(* Logix 5000 project; controller Close_Palletizing 1769-L33ERM rev 33.13; software revision 33.00 *)

TASK MainTask (continuous, watchdog 500 ms) : MainProgram

MODULES
   Local : 1769-L33ERM (Compact 0, rev 33.13)
      BrazingOvenEthernetCard : 1756-ENBT (Ethernet 192.168.1.100, rev 5.1, Output RPI 10 ms)
         BrazingOvenPLC : vendor 1 type 14 code 92 (ICP 0, rev 23.12, $5738e604$ RPI 20 ms, $87ed6ff7$ RPI 20 ms)
      Fanuc_5 : ETHERNET-MODULE (Ethernet 192.168.1.5, rev 1.1, Output RPI 10 ms)
           Fanuc_5:O.Data[3].1   // *Hold
           Fanuc_5:O.Data[0]   // Part Width to give to Fanuc
           Fanuc_5:O.Data[2]   // Part Length to give to Fanuc
           Fanuc_5:O.Data[3].0   // *IMSTP
           Fanuc_5:O.Data[1]   // Part ID to give to Fanuc
           Fanuc_5:O.Data[3].2   // *SFSPD
           Fanuc_5:O.Data[3].3   // Cycle stop
           Fanuc_5:O.Data[3].4   // Fault reset
           Fanuc_5:O.Data[3].5   // Start
           Fanuc_5:O.Data[3].6   // Home
           Fanuc_5:O.Data[3].7   // Enable
           Fanuc_5:O.Data[3].8   // PNS strobe
           Fanuc_5:O.Data[3].9   // Prod start
           Fanuc_5:I.Data[2].0   // Cmd enabled
           Fanuc_5:I.Data[2].1   // System ready
           Fanuc_5:I.Data[2].2   // Prg running
           Fanuc_5:I.Data[2].3   // Prg paused
           Fanuc_5:I.Data[2].4   // Motion held
           Fanuc_5:I.Data[2].5   // Fault
           Fanuc_5:I.Data[2].6   // At perch
           Fanuc_5:I.Data[2].7   // TP enabled
           Fanuc_5:I.Data[2].8   // Batt alarm
           Fanuc_5:I.Data[2].9   // Busy
           Fanuc_5:I.Data[2].10   // ACK1/SNO1
           Fanuc_5:I.Data[2].11   // ACK2/SNO2
           Fanuc_5:I.Data[2].12   // ACK3/SNO3
           Fanuc_5:I.Data[2].13   // ACK4/SNO4
           Fanuc_5:I.Data[2].14   // ACK5/SNO5
           Fanuc_5:I.Data[2].15   // ACK6/SNO6
           Fanuc_5:I.Data[3].2   // SNACK
           Fanuc_5:I.Data[3].0   // ACK7/SNO7
           Fanuc_5:I.Data[3].1   // ACK8/SNO8
           Fanuc_5:I.Data[3].3   // Reserved
      YRC1000_Rbt_Ctlr : ETHERNET-MODULE (Ethernet 192.168.1.41, rev 1.1, Output RPI 10 ms)
      IFM_Module_Fence : vendor 322 type 12 code 1120 (Ethernet 192.168.1.43, rev 1.5, StandardDataDriven RPI 10 ms)
           IFM_Module_Fence:I1.Data[0].0   // Port 1 Pin 4
           IFM_Module_Fence:I1.Data[0].1   // Port 2 Pin 4
           IFM_Module_Fence:I1.Data[0].10   // Port 3 Pin 2
           IFM_Module_Fence:I1.Data[0].11   // Port 4 Pin 2
           IFM_Module_Fence:I1.Data[0].12   // Reserved
           IFM_Module_Fence:I1.Data[0].13   // Reserved
           IFM_Module_Fence:I1.Data[0].14   // Reserved
           IFM_Module_Fence:I1.Data[0].15   // Reserved
           IFM_Module_Fence:I1.Data[0].2   // Port 3 Pin 4
           IFM_Module_Fence:I1.Data[0].3   // Port 4 Pin 4
           IFM_Module_Fence:I1.Data[0].4   // Reserved
           IFM_Module_Fence:I1.Data[0].5   // Reserved
           IFM_Module_Fence:I1.Data[0].6   // Reserved
           IFM_Module_Fence:I1.Data[0].7   // Reserved
           IFM_Module_Fence:I1.Data[0].8   // Port 1 Pin 2
           IFM_Module_Fence:I1.Data[0].9   // Port 2 Pin 2
           IFM_Module_Fence:I1.Data[100]   // Port 3 Input Process Data
           IFM_Module_Fence:I1.Data[101]   // Port 3 Input Process Data
           IFM_Module_Fence:I1.Data[102]   // Port 3 Input Process Data
           IFM_Module_Fence:I1.Data[103]   // Port 3 Input Process Data
           IFM_Module_Fence:I1.Data[104]   // Port 3 Input Process Data
           IFM_Module_Fence:I1.Data[105]   // Port 3 Input Process Data
           IFM_Module_Fence:I1.Data[106]   // Port 3 Input Process Data
           IFM_Module_Fence:I1.Data[107]   // Port 4 Input Process Data
           IFM_Module_Fence:I1.Data[108]   // Port 4 Input Process Data
           IFM_Module_Fence:I1.Data[109]   // Port 4 Input Process Data
           IFM_Module_Fence:I1.Data[10]   // Command Response Or Diagnostic Data 7
           IFM_Module_Fence:I1.Data[110]   // Port 4 Input Process Data
           IFM_Module_Fence:I1.Data[111]   // Port 4 Input Process Data
           IFM_Module_Fence:I1.Data[112]   // Port 4 Input Process Data
           IFM_Module_Fence:I1.Data[113]   // Port 4 Input Process Data
           IFM_Module_Fence:I1.Data[114]   // Port 4 Input Process Data
           IFM_Module_Fence:I1.Data[115]   // Port 4 Input Process Data
           IFM_Module_Fence:I1.Data[116]   // Port 4 Input Process Data
           IFM_Module_Fence:I1.Data[117]   // Port 4 Input Process Data
           IFM_Module_Fence:I1.Data[118]   // Port 4 Input Process Data
           IFM_Module_Fence:I1.Data[119]   // Port 4 Input Process Data
           IFM_Module_Fence:I1.Data[11]   // Command Response Or Diagnostic Data 9
           IFM_Module_Fence:I1.Data[120]   // Port 4 Input Process Data
           IFM_Module_Fence:I1.Data[121]   // Port 4 Input Process Data
           IFM_Module_Fence:I1.Data[122]   // Port 4 Input Process Data
           IFM_Module_Fence:I1.Data[12]   // Command Response Or Diagnostic Data 11
           IFM_Module_Fence:I1.Data[13]   // Command Response Or Diagnostic Data 13
           IFM_Module_Fence:I1.Data[14]   // Command Response Or Diagnostic Data 15
           IFM_Module_Fence:I1.Data[15]   // Command Response Or Diagnostic Data 17
           IFM_Module_Fence:I1.Data[16]   // Command Response Or Diagnostic Data 19
           IFM_Module_Fence:I1.Data[17]   // Command Response Or Diagnostic Data 21
           IFM_Module_Fence:I1.Data[18]   // Command Response Or Diagnostic Data 23
           IFM_Module_Fence:I1.Data[19]   // Command Response Or Diagnostic Data 25
           IFM_Module_Fence:I1.Data[1]   // AL1x2x Digital Input Short/Overload Status
           IFM_Module_Fence:I1.Data[1].0   // Port 1 Short/Overload
           IFM_Module_Fence:I1.Data[1].1   // Port 2 Short/Overload
           IFM_Module_Fence:I1.Data[1].10   // Reserved
           IFM_Module_Fence:I1.Data[1].11   // Reserved
           IFM_Module_Fence:I1.Data[1].12   // Reserved
           IFM_Module_Fence:I1.Data[1].13   // Reserved
           IFM_Module_Fence:I1.Data[1].14   // Reserved
           IFM_Module_Fence:I1.Data[1].15   // Reserved
           IFM_Module_Fence:I1.Data[1].2   // Port 3 Short/Overload
           IFM_Module_Fence:I1.Data[1].3   // Port 4 Short/Overload
           IFM_Module_Fence:I1.Data[1].4   // Reserved
           IFM_Module_Fence:I1.Data[1].5   // Reserved
           IFM_Module_Fence:I1.Data[1].6   // Reserved
           IFM_Module_Fence:I1.Data[1].7   // Reserved
           IFM_Module_Fence:I1.Data[1].8   // Reserved
           IFM_Module_Fence:I1.Data[1].9   // Reserved
           IFM_Module_Fence:I1.Data[20]   // Command Response Or Diagnostic Data 27
           IFM_Module_Fence:I1.Data[21]   // Command Response Or Diagnostic Data 29
           IFM_Module_Fence:I1.Data[22]   // Command Response Or Diagnostic Data 31
           IFM_Module_Fence:I1.Data[23].0   // Port 1 IO-Link Mode
           IFM_Module_Fence:I1.Data[23].1   // Port 1 NO IO-Link Device Connected
           IFM_Module_Fence:I1.Data[23].10   // Reserved
           IFM_Module_Fence:I1.Data[23].11   // Reserved
           IFM_Module_Fence:I1.Data[23].12   // Reserved
           IFM_Module_Fence:I1.Data[23].13   // Reserved
           IFM_Module_Fence:I1.Data[23].14   // Reserved
           IFM_Module_Fence:I1.Data[23].15   // Reserved
           IFM_Module_Fence:I1.Data[23].2   // Port 1 IO-Link Data Invalid
           IFM_Module_Fence:I1.Data[23].3   // Port 1 Incorrect Vendor or Device ID
           IFM_Module_Fence:I1.Data[23].5   // Reserved
           IFM_Module_Fence:I1.Data[23].6   // Reserved
           IFM_Module_Fence:I1.Data[23].7   // Reserved
           IFM_Module_Fence:I1.Data[23].8   // Reserved
           IFM_Module_Fence:I1.Data[23].9   // Reserved
           IFM_Module_Fence:I1.Data[24]   // Port 1 Vendor ID
           IFM_Module_Fence:I1.Data[25]   // Port 1 Device ID (Low Word)
           IFM_Module_Fence:I1.Data[26]   // Port 1 Device ID (High Word)
           IFM_Module_Fence:I1.Data[0]   // AL1x2x Digital Input Status
           IFM_Module_Fence:I1.Data[27]   // Port 1 IO-Link Event Data
           IFM_Module_Fence:I1.Data[27].0   // Port 1 Event Instance
           IFM_Module_Fence:I1.Data[27].1   // Port 1 Event Instance
           IFM_Module_Fence:I1.Data[27].10   // Port 1 Event Code 1
           IFM_Module_Fence:I1.Data[27].11   // Port 1 Event Code 1
           IFM_Module_Fence:I1.Data[27].12   // Port 1 Event Code 1
           IFM_Module_Fence:I1.Data[27].13   // Port 1 Event Code 1
           IFM_Module_Fence:I1.Data[27].14   // Port 1 Event Code 1
           IFM_Module_Fence:I1.Data[27].15   // Port 1 Event Code 1
           IFM_Module_Fence:I1.Data[27].3   // Port 1 Event Source
           IFM_Module_Fence:I1.Data[27].8   // Port 1 Event Code 1
           IFM_Module_Fence:I1.Data[27].9   // Port 1 Event Code 1
           IFM_Module_Fence:I1.Data[28].0   // Port 1 Event Code 2
           IFM_Module_Fence:I1.Data[28].1   // Port 1 Event Code 2
           IFM_Module_Fence:I1.Data[28].10   // Port 1 Event Instance
           IFM_Module_Fence:I1.Data[27].2   // Port 1 Event Instance
           IFM_Module_Fence:I1.Data[28].12   // Port 1 Event Type
           IFM_Module_Fence:I1.Data[28].13   // Port 1 Event Type
           IFM_Module_Fence:I1.Data[28].14   // Port 1 Event Mode
           IFM_Module_Fence:I1.Data[28].15   // Port 1 Event Mode
           IFM_Module_Fence:I1.Data[28].2   // Port 1 Event Code 2
           IFM_Module_Fence:I1.Data[28].3   // Port 1 Event Code 2
           IFM_Module_Fence:I1.Data[28].4   // Port 1 Event Code 2
           IFM_Module_Fence:I1.Data[28].5   // Port 1 Event Code 2
           IFM_Module_Fence:I1.Data[28].6   // Port 1 Event Code 2
           IFM_Module_Fence:I1.Data[28].7   // Port 1 Event Code 2
           IFM_Module_Fence:I1.Data[28].11   // Port 1 Event Source
           IFM_Module_Fence:I1.Data[28].8   // Port 1 Event Instance
           IFM_Module_Fence:I1.Data[28].9   // Port 1 Event Instance
           IFM_Module_Fence:I1.Data[29].0   // Port 1 Event Code 1
           IFM_Module_Fence:I1.Data[29].1   // Port 1 Event Code 1
           IFM_Module_Fence:I1.Data[29]   // Port 1 IO-Link Event Data
           IFM_Module_Fence:I1.Data[29].10   // Port 1 Event Code 2
           IFM_Module_Fence:I1.Data[29].11   // Port 1 Event Code 2
           IFM_Module_Fence:I1.Data[29].12   // Port 1 Event Code 2
           IFM_Module_Fence:I1.Data[29].13   // Port 1 Event Code 2
           IFM_Module_Fence:I1.Data[29].14   // Port 1 Event Code 2
           IFM_Module_Fence:I1.Data[29].2   // Port 1 Event Code 1
           IFM_Module_Fence:I1.Data[29].3   // Port 1 Event Code 1
           IFM_Module_Fence:I1.Data[29].4   // Port 1 Event Code 1
           IFM_Module_Fence:I1.Data[29].5   // Port 1 Event Code 1
           IFM_Module_Fence:I1.Data[29].6   // Port 1 Event Code 1
           IFM_Module_Fence:I1.Data[29].7   // Port 1 Event Code 1
           IFM_Module_Fence:I1.Data[29].8   // Port 1 Event Code 2
           IFM_Module_Fence:I1.Data[29].9   // Port 1 Event Code 2
           IFM_Module_Fence:I1.Data[2]   // Port Number
           IFM_Module_Fence:I1.Data[29].15   // Port 1 Event Code 2
           IFM_Module_Fence:I1.Data[30]   // Port 1 IO-Link Event Data
           IFM_Module_Fence:I1.Data[30].0   // Port 1 Event Instance
           IFM_Module_Fence:I1.Data[30].1   // Port 1 Event Instance
           IFM_Module_Fence:I1.Data[30].10   // Port 1 Event Code 1
           IFM_Module_Fence:I1.Data[30].11   // Port 1 Event Code 1
           IFM_Module_Fence:I1.Data[30].12   // Port 1 Event Code 1
           IFM_Module_Fence:I1.Data[30].13   // Port 1 Event Code 1
           IFM_Module_Fence:I1.Data[30].14   // Port 1 Event Code 1
           IFM_Module_Fence:I1.Data[30].15   // Port 1 Event Code 1
           IFM_Module_Fence:I1.Data[30].3   // Port 1 Event Source
           IFM_Module_Fence:I1.Data[23]   // Port 1 IO Link Status
           IFM_Module_Fence:I1.Data[27].4   // Port 1 Event Type
           IFM_Module_Fence:I1.Data[27].5   // Port 1 Event Type
           IFM_Module_Fence:I1.Data[27].6   // Port 1 Event Mode
           IFM_Module_Fence:I1.Data[30].8   // Port 1 Event Code 1
           IFM_Module_Fence:I1.Data[30].9   // Port 1 Event Code 1
           IFM_Module_Fence:I1.Data[30].2   // Port 1 Event Instance
           IFM_Module_Fence:I1.Data[31].0   // Port 1 Event Code 2
           IFM_Module_Fence:I1.Data[31].1   // Port 1 Event Code 2
           IFM_Module_Fence:I1.Data[31].10   // Reserved
           IFM_Module_Fence:I1.Data[31].11   // Reserved
           IFM_Module_Fence:I1.Data[31].12   // Reserved
           IFM_Module_Fence:I1.Data[31].13   // Reserved
           IFM_Module_Fence:I1.Data[31].14   // Reserved
           IFM_Module_Fence:I1.Data[31].15   // Reserved
           IFM_Module_Fence:I1.Data[31].2   // Port 1 Event Code 2
           IFM_Module_Fence:I1.Data[31].3   // Port 1 Event Code 2
           IFM_Module_Fence:I1.Data[31].4   // Port 1 Event Code 2
           IFM_Module_Fence:I1.Data[31].5   // Port 1 Event Code 2
           IFM_Module_Fence:I1.Data[31].6   // Port 1 Event Code 2
           IFM_Module_Fence:I1.Data[31].7   // Port 1 Event Code 2
           IFM_Module_Fence:I1.Data[31].8   // Reserved
           IFM_Module_Fence:I1.Data[31].9   // Reserved
           IFM_Module_Fence:I1.Data[27].7   // Port 1 Event Mode
           IFM_Module_Fence:I1.Data[32].0   // Port 2 IO-Link Mode
           IFM_Module_Fence:I1.Data[32].1   // Port 2 NO IO-Link Device Connected
           IFM_Module_Fence:I1.Data[32].10   // Reserved
           IFM_Module_Fence:I1.Data[32].11   // Reserved
           IFM_Module_Fence:I1.Data[32].12   // Reserved
           IFM_Module_Fence:I1.Data[32].13   // Reserved
           IFM_Module_Fence:I1.Data[32].14   // Reserved
           IFM_Module_Fence:I1.Data[32].15   // Reserved
           IFM_Module_Fence:I1.Data[32].2   // Port 2 IO-Link Data Invalid
           IFM_Module_Fence:I1.Data[32].3   // Port 2 Incorrect Vendor or Device ID
           IFM_Module_Fence:I1.Data[23].4   // Port 1 IO-Link Data String Error
           IFM_Module_Fence:I1.Data[32].5   // Reserved
           IFM_Module_Fence:I1.Data[32].6   // Reserved
           IFM_Module_Fence:I1.Data[32].7   // Reserved
           IFM_Module_Fence:I1.Data[32].8   // Reserved
           IFM_Module_Fence:I1.Data[32].9   // Reserved
           IFM_Module_Fence:I1.Data[33]   // Port 2 Vendor ID
           IFM_Module_Fence:I1.Data[34]   // Port 2 Device ID (Low Word)
           IFM_Module_Fence:I1.Data[35]   // Port 2 Device ID (High Word)
           IFM_Module_Fence:I1.Data[31]   // Port 1 IO-Link Event Data
           IFM_Module_Fence:I1.Data[36]   // Port 2 IO-Link Event Data
           IFM_Module_Fence:I1.Data[36].0   // Port 2 Event Instance
           IFM_Module_Fence:I1.Data[36].1   // Port 2 Event Instance
           IFM_Module_Fence:I1.Data[36].10   // Port 2 Event Code 1
           IFM_Module_Fence:I1.Data[36].11   // Port 2 Event Code 1
           IFM_Module_Fence:I1.Data[36].12   // Port 2 Event Code 1
           IFM_Module_Fence:I1.Data[36].13   // Port 2 Event Code 1
           IFM_Module_Fence:I1.Data[36].14   // Port 2 Event Code 1
           IFM_Module_Fence:I1.Data[36].15   // Port 2 Event Code 1
           IFM_Module_Fence:I1.Data[36].3   // Port 2 Event Source
           IFM_Module_Fence:I1.Data[30].4   // Port 1 Event Type
           IFM_Module_Fence:I1.Data[30].5   // Port 1 Event Type
           IFM_Module_Fence:I1.Data[30].6   // Port 1 Event Mode
           IFM_Module_Fence:I1.Data[30].7   // Port 1 Event Mode
           IFM_Module_Fence:I1.Data[36].8   // Port 2 Event Code 1
           IFM_Module_Fence:I1.Data[36].9   // Port 2 Event Code 1
           IFM_Module_Fence:I1.Data[28]   // Port 1 IO-Link Event Data
           IFM_Module_Fence:I1.Data[37].0   // Port 2 Event Code 2
           IFM_Module_Fence:I1.Data[37].1   // Port 2 Event Code 2
           IFM_Module_Fence:I1.Data[37].10   // Port 2 Event Instance
           IFM_Module_Fence:I1.Data[36].2   // Port 2 Event Instance
           IFM_Module_Fence:I1.Data[37].12   // Port 2 Event Type
           IFM_Module_Fence:I1.Data[37].13   // Port 2 Event Type
           IFM_Module_Fence:I1.Data[37].14   // Port 2 Event Mode
           IFM_Module_Fence:I1.Data[37].15   // Port 2 Event Mode
           IFM_Module_Fence:I1.Data[37].2   // Port 2 Event Code 2
           IFM_Module_Fence:I1.Data[37].3   // Port 2 Event Code 2
           IFM_Module_Fence:I1.Data[37].4   // Port 2 Event Code 2
           IFM_Module_Fence:I1.Data[37].5   // Port 2 Event Code 2
           IFM_Module_Fence:I1.Data[37].6   // Port 2 Event Code 2
           IFM_Module_Fence:I1.Data[37].7   // Port 2 Event Code 2
           IFM_Module_Fence:I1.Data[37].11   // Port 2 Event Source
           IFM_Module_Fence:I1.Data[37].8   // Port 2 Event Instance
           IFM_Module_Fence:I1.Data[37].9   // Port 2 Event Instance
           IFM_Module_Fence:I1.Data[38].0   // Port 2 Event Code 1
           IFM_Module_Fence:I1.Data[38].1   // Port 2 Event Code 1
           IFM_Module_Fence:I1.Data[38]   // Port 2 IO-Link Event Data
           IFM_Module_Fence:I1.Data[38].10   // Port 2 Event Code 2
           IFM_Module_Fence:I1.Data[38].11   // Port 2 Event Code 2
           IFM_Module_Fence:I1.Data[38].12   // Port 2 Event Code 2
           IFM_Module_Fence:I1.Data[38].13   // Port 2 Event Code 2
           IFM_Module_Fence:I1.Data[38].14   // Port 2 Event Code 2
           IFM_Module_Fence:I1.Data[38].2   // Port 2 Event Code 1
           IFM_Module_Fence:I1.Data[38].3   // Port 2 Event Code 1
           IFM_Module_Fence:I1.Data[38].4   // Port 2 Event Code 1
           IFM_Module_Fence:I1.Data[38].5   // Port 2 Event Code 1
           IFM_Module_Fence:I1.Data[38].6   // Port 2 Event Code 1
           IFM_Module_Fence:I1.Data[38].7   // Port 2 Event Code 1
           IFM_Module_Fence:I1.Data[38].8   // Port 2 Event Code 2
           IFM_Module_Fence:I1.Data[38].9   // Port 2 Event Code 2
           IFM_Module_Fence:I1.Data[38].15   // Port 2 Event Code 2
           IFM_Module_Fence:I1.Data[39]   // Port 2 IO-Link Event Data
           IFM_Module_Fence:I1.Data[39].0   // Port 2 Event Instance
           IFM_Module_Fence:I1.Data[39].1   // Port 2 Event Instance
           IFM_Module_Fence:I1.Data[39].10   // Port 2 Event Code 1
           IFM_Module_Fence:I1.Data[39].11   // Port 2 Event Code 1
           IFM_Module_Fence:I1.Data[39].12   // Port 2 Event Code 1
           IFM_Module_Fence:I1.Data[39].13   // Port 2 Event Code 1
           IFM_Module_Fence:I1.Data[39].14   // Port 2 Event Code 1
           IFM_Module_Fence:I1.Data[39].15   // Port 2 Event Code 1
           IFM_Module_Fence:I1.Data[39].3   // Port 2 Event Source
           IFM_Module_Fence:I1.Data[32]   // Port 2 IO Link Status
           IFM_Module_Fence:I1.Data[36].4   // Port 2 Event Type
           IFM_Module_Fence:I1.Data[36].5   // Port 2 Event Type
           IFM_Module_Fence:I1.Data[36].6   // Port 2 Event Mode
           IFM_Module_Fence:I1.Data[39].8   // Port 2 Event Code 1
           IFM_Module_Fence:I1.Data[39].9   // Port 2 Event Code 1
           IFM_Module_Fence:I1.Data[3]   // Index Number
           IFM_Module_Fence:I1.Data[39].2   // Port 2 Event Instance
           IFM_Module_Fence:I1.Data[40].0   // Port 2 Event Code 2
           IFM_Module_Fence:I1.Data[40].1   // Port 2 Event Code 2
           IFM_Module_Fence:I1.Data[40].10   // Reserved
           IFM_Module_Fence:I1.Data[40].11   // Reserved
           IFM_Module_Fence:I1.Data[40].12   // Reserved
           IFM_Module_Fence:I1.Data[40].13   // Reserved
           IFM_Module_Fence:I1.Data[40].14   // Reserved
           IFM_Module_Fence:I1.Data[40].15   // Reserved
           IFM_Module_Fence:I1.Data[40].2   // Port 2 Event Code 2
           IFM_Module_Fence:I1.Data[40].3   // Port 2 Event Code 2
           IFM_Module_Fence:I1.Data[40].4   // Port 2 Event Code 2
           IFM_Module_Fence:I1.Data[40].5   // Port 2 Event Code 2
           IFM_Module_Fence:I1.Data[40].6   // Port 2 Event Code 2
           IFM_Module_Fence:I1.Data[40].7   // Port 2 Event Code 2
           IFM_Module_Fence:I1.Data[40].8   // Reserved
           IFM_Module_Fence:I1.Data[40].9   // Reserved
           IFM_Module_Fence:I1.Data[36].7   // Port 2 Event Mode
           IFM_Module_Fence:I1.Data[41].0   // Port 3 IO-Link Mode
           IFM_Module_Fence:I1.Data[41].1   // Port 3 NO IO-Link Device Connected
           IFM_Module_Fence:I1.Data[41].10   // Reserved
           IFM_Module_Fence:I1.Data[41].11   // Reserved
           IFM_Module_Fence:I1.Data[41].12   // Reserved
           IFM_Module_Fence:I1.Data[41].13   // Reserved
           IFM_Module_Fence:I1.Data[41].14   // Reserved
           IFM_Module_Fence:I1.Data[41].15   // Reserved
           IFM_Module_Fence:I1.Data[41].2   // Port 3 IO-Link Data Invalid
           IFM_Module_Fence:I1.Data[41].3   // Port 3 Incorrect Vendor or Device ID
           IFM_Module_Fence:I1.Data[32].4   // Port 2 IO-Link Data String Error
           IFM_Module_Fence:I1.Data[41].5   // Reserved
           IFM_Module_Fence:I1.Data[41].6   // Reserved
           IFM_Module_Fence:I1.Data[41].7   // Reserved
           IFM_Module_Fence:I1.Data[41].8   // Reserved
           IFM_Module_Fence:I1.Data[41].9   // Reserved
           IFM_Module_Fence:I1.Data[42]   // Port 3 Vendor ID
           IFM_Module_Fence:I1.Data[43]   // Port 3 Device ID (Low Word)
           IFM_Module_Fence:I1.Data[44]   // Port 3 Device ID (High Word)
           IFM_Module_Fence:I1.Data[40]   // Port 2 IO-Link Event Data
           IFM_Module_Fence:I1.Data[45]   // Port 3 IO-Link Event Data
           IFM_Module_Fence:I1.Data[45].0   // Port 3 Event Instance
           IFM_Module_Fence:I1.Data[45].1   // Port 3 Event Instance
           IFM_Module_Fence:I1.Data[45].10   // Port 3 Event Code 1
           IFM_Module_Fence:I1.Data[45].11   // Port 3 Event Code 1
           IFM_Module_Fence:I1.Data[45].12   // Port 3 Event Code 1
           IFM_Module_Fence:I1.Data[45].13   // Port 3 Event Code 1
           IFM_Module_Fence:I1.Data[45].14   // Port 3 Event Code 1
           IFM_Module_Fence:I1.Data[45].15   // Port 3 Event Code 1
           IFM_Module_Fence:I1.Data[45].3   // Port 3 Event Source
           IFM_Module_Fence:I1.Data[39].4   // Port 2 Event Type
           IFM_Module_Fence:I1.Data[39].5   // Port 2 Event Type
           IFM_Module_Fence:I1.Data[39].6   // Port 2 Event Mode
           IFM_Module_Fence:I1.Data[39].7   // Port 2 Event Mode
           IFM_Module_Fence:I1.Data[45].8   // Port 3 Event Code 1
           IFM_Module_Fence:I1.Data[45].9   // Port 3 Event Code 1
           IFM_Module_Fence:I1.Data[37]   // Port 2 IO-Link Event Data
           IFM_Module_Fence:I1.Data[46].0   // Port 3 Event Code 2
           IFM_Module_Fence:I1.Data[46].1   // Port 3 Event Code 2
           IFM_Module_Fence:I1.Data[46].10   // Port 3 Event Instance
           IFM_Module_Fence:I1.Data[45].2   // Port 3 Event Instance
           IFM_Module_Fence:I1.Data[46].12   // Port 3 Event Type
           IFM_Module_Fence:I1.Data[46].13   // Port 3 Event Type
           IFM_Module_Fence:I1.Data[46].14   // Port 3 Event Mode
           IFM_Module_Fence:I1.Data[46].15   // Port 3 Event Mode
           IFM_Module_Fence:I1.Data[46].2   // Port 3 Event Code 2
           IFM_Module_Fence:I1.Data[46].3   // Port 3 Event Code 2
           IFM_Module_Fence:I1.Data[46].4   // Port 3 Event Code 2
           IFM_Module_Fence:I1.Data[46].5   // Port 3 Event Code 2
           IFM_Module_Fence:I1.Data[46].6   // Port 3 Event Code 2
           IFM_Module_Fence:I1.Data[46].7   // Port 3 Event Code 2
           IFM_Module_Fence:I1.Data[46].11   // Port 3 Event Source
           IFM_Module_Fence:I1.Data[46].8   // Port 3 Event Instance
           IFM_Module_Fence:I1.Data[46].9   // Port 3 Event Instance
           IFM_Module_Fence:I1.Data[47].0   // Port 3 Event Code 1
           IFM_Module_Fence:I1.Data[47].1   // Port 3 Event Code 1
           IFM_Module_Fence:I1.Data[47]   // Port 3 IO-Link Event Data
           IFM_Module_Fence:I1.Data[47].10   // Port 3 Event Code 2
           IFM_Module_Fence:I1.Data[47].11   // Port 3 Event Code 2
           IFM_Module_Fence:I1.Data[47].12   // Port 3 Event Code 2
           IFM_Module_Fence:I1.Data[47].13   // Port 3 Event Code 2
           IFM_Module_Fence:I1.Data[47].14   // Port 3 Event Code 2
           IFM_Module_Fence:I1.Data[47].2   // Port 3 Event Code 1
           IFM_Module_Fence:I1.Data[47].3   // Port 3 Event Code 1
           IFM_Module_Fence:I1.Data[47].4   // Port 3 Event Code 1
           IFM_Module_Fence:I1.Data[47].5   // Port 3 Event Code 1
           IFM_Module_Fence:I1.Data[47].6   // Port 3 Event Code 1
           IFM_Module_Fence:I1.Data[47].7   // Port 3 Event Code 1
           IFM_Module_Fence:I1.Data[47].8   // Port 3 Event Code 2
           IFM_Module_Fence:I1.Data[47].9   // Port 3 Event Code 2
           IFM_Module_Fence:I1.Data[47].15   // Port 3 Event Code 2
           IFM_Module_Fence:I1.Data[48]   // Port 3 IO-Link Event Data
           IFM_Module_Fence:I1.Data[48].0   // Port 3 Event Instance
           IFM_Module_Fence:I1.Data[48].1   // Port 3 Event Instance
           IFM_Module_Fence:I1.Data[48].10   // Port 3 Event Code 1
           IFM_Module_Fence:I1.Data[48].11   // Port 3 Event Code 1
           IFM_Module_Fence:I1.Data[48].12   // Port 3 Event Code 1
           IFM_Module_Fence:I1.Data[48].13   // Port 3 Event Code 1
           IFM_Module_Fence:I1.Data[48].14   // Port 3 Event Code 1
           IFM_Module_Fence:I1.Data[48].15   // Port 3 Event Code 1
           IFM_Module_Fence:I1.Data[48].3   // Port 3 Event Source
           IFM_Module_Fence:I1.Data[41]   // Port 3 IO Link Status
           IFM_Module_Fence:I1.Data[45].4   // Port 3 Event Type
           IFM_Module_Fence:I1.Data[45].5   // Port 3 Event Type
           IFM_Module_Fence:I1.Data[45].6   // Port 3 Event Mode
           IFM_Module_Fence:I1.Data[48].8   // Port 3 Event Code 1
           IFM_Module_Fence:I1.Data[48].9   // Port 3 Event Code 1
           IFM_Module_Fence:I1.Data[48].2   // Port 3 Event Instance
           IFM_Module_Fence:I1.Data[49].0   // Port 3 Event Code 2
           IFM_Module_Fence:I1.Data[49].1   // Port 3 Event Code 2
           IFM_Module_Fence:I1.Data[49].10   // Reserved
           IFM_Module_Fence:I1.Data[49].11   // Reserved
           IFM_Module_Fence:I1.Data[49].12   // Reserved
           IFM_Module_Fence:I1.Data[49].13   // Reserved
           IFM_Module_Fence:I1.Data[49].14   // Reserved
           IFM_Module_Fence:I1.Data[49].15   // Reserved
           IFM_Module_Fence:I1.Data[49].2   // Port 3 Event Code 2
           IFM_Module_Fence:I1.Data[49].3   // Port 3 Event Code 2
           IFM_Module_Fence:I1.Data[49].4   // Port 3 Event Code 2
           IFM_Module_Fence:I1.Data[49].5   // Port 3 Event Code 2
           IFM_Module_Fence:I1.Data[49].6   // Port 3 Event Code 2
           IFM_Module_Fence:I1.Data[49].7   // Port 3 Event Code 2
           IFM_Module_Fence:I1.Data[49].8   // Reserved
           IFM_Module_Fence:I1.Data[49].9   // Reserved
           IFM_Module_Fence:I1.Data[4]   // SubIndex Number
           IFM_Module_Fence:I1.Data[45].7   // Port 3 Event Mode
           IFM_Module_Fence:I1.Data[50].0   // Port 4 IO-Link Mode
           IFM_Module_Fence:I1.Data[50].1   // Port 4 NO IO-Link Device Connected
           IFM_Module_Fence:I1.Data[50].10   // Reserved
           IFM_Module_Fence:I1.Data[50].11   // Reserved
           IFM_Module_Fence:I1.Data[50].12   // Reserved
           IFM_Module_Fence:I1.Data[50].13   // Reserved
           IFM_Module_Fence:I1.Data[50].14   // Reserved
           IFM_Module_Fence:I1.Data[50].15   // Reserved
           IFM_Module_Fence:I1.Data[50].2   // Port 4 IO-Link Data Invalid
           IFM_Module_Fence:I1.Data[50].3   // Port 4 Incorrect Vendor or Device ID
           IFM_Module_Fence:I1.Data[41].4   // Port 3 IO-Link Data String Error
           IFM_Module_Fence:I1.Data[50].5   // Reserved
           IFM_Module_Fence:I1.Data[50].6   // Reserved
           IFM_Module_Fence:I1.Data[50].7   // Reserved
           IFM_Module_Fence:I1.Data[50].8   // Reserved
           IFM_Module_Fence:I1.Data[50].9   // Reserved
           IFM_Module_Fence:I1.Data[51]   // Port 4 Vendor ID
           IFM_Module_Fence:I1.Data[52]   // Port 4 Device ID (Low Word)
           IFM_Module_Fence:I1.Data[53]   // Port 4 Device ID (High Word)
           IFM_Module_Fence:I1.Data[49]   // Port 3 IO-Link Event Data
           IFM_Module_Fence:I1.Data[54]   // Port 4 IO-Link Event Data
           IFM_Module_Fence:I1.Data[54].0   // Port 4 Event Instance
           IFM_Module_Fence:I1.Data[54].1   // Port 4 Event Instance
           IFM_Module_Fence:I1.Data[54].10   // Port 4 Event Code 1
           IFM_Module_Fence:I1.Data[54].11   // Port 4 Event Code 1
           IFM_Module_Fence:I1.Data[54].12   // Port 4 Event Code 1
           IFM_Module_Fence:I1.Data[54].13   // Port 4 Event Code 1
           IFM_Module_Fence:I1.Data[54].14   // Port 4 Event Code 1
           IFM_Module_Fence:I1.Data[54].15   // Port 4 Event Code 1
           IFM_Module_Fence:I1.Data[54].3   // Port 4 Event Source
           IFM_Module_Fence:I1.Data[48].4   // Port 3 Event Type
           IFM_Module_Fence:I1.Data[48].5   // Port 3 Event Type
           IFM_Module_Fence:I1.Data[48].6   // Port 3 Event Mode
           IFM_Module_Fence:I1.Data[48].7   // Port 3 Event Mode
           IFM_Module_Fence:I1.Data[54].8   // Port 4 Event Code 1
           IFM_Module_Fence:I1.Data[54].9   // Port 4 Event Code 1
           IFM_Module_Fence:I1.Data[46]   // Port 3 IO-Link Event Data
           IFM_Module_Fence:I1.Data[55].0   // Port 4 Event Code 2
           IFM_Module_Fence:I1.Data[55].1   // Port 4 Event Code 2
           IFM_Module_Fence:I1.Data[55].10   // Port 4 Event Instance
           IFM_Module_Fence:I1.Data[54].2   // Port 4 Event Instance
           IFM_Module_Fence:I1.Data[55].12   // Port 4 Event Type
           IFM_Module_Fence:I1.Data[55].13   // Port 4 Event Type
           IFM_Module_Fence:I1.Data[55].14   // Port 4 Event Mode
           IFM_Module_Fence:I1.Data[55].15   // Port 4 Event Mode
           IFM_Module_Fence:I1.Data[55].2   // Port 4 Event Code 2
           IFM_Module_Fence:I1.Data[55].3   // Port 4 Event Code 2
           IFM_Module_Fence:I1.Data[55].4   // Port 4 Event Code 2
           IFM_Module_Fence:I1.Data[55].5   // Port 4 Event Code 2
           IFM_Module_Fence:I1.Data[55].6   // Port 4 Event Code 2
           IFM_Module_Fence:I1.Data[55].7   // Port 4 Event Code 2
           IFM_Module_Fence:I1.Data[55].11   // Port 4 Event Source
           IFM_Module_Fence:I1.Data[55].8   // Port 4 Event Instance
           IFM_Module_Fence:I1.Data[55].9   // Port 4 Event Instance
           IFM_Module_Fence:I1.Data[56].0   // Port 4 Event Code 1
           IFM_Module_Fence:I1.Data[56].1   // Port 4 Event Code 1
           IFM_Module_Fence:I1.Data[56]   // Port 4 IO-Link Event Data
           IFM_Module_Fence:I1.Data[56].10   // Port 4 Event Code 2
           IFM_Module_Fence:I1.Data[56].11   // Port 4 Event Code 2
           IFM_Module_Fence:I1.Data[56].12   // Port 4 Event Code 2
           IFM_Module_Fence:I1.Data[56].13   // Port 4 Event Code 2
           IFM_Module_Fence:I1.Data[56].14   // Port 4 Event Code 2
           IFM_Module_Fence:I1.Data[56].2   // Port 4 Event Code 1
           IFM_Module_Fence:I1.Data[56].3   // Port 4 Event Code 1
           IFM_Module_Fence:I1.Data[56].4   // Port 4 Event Code 1
           IFM_Module_Fence:I1.Data[56].5   // Port 4 Event Code 1
           IFM_Module_Fence:I1.Data[56].6   // Port 4 Event Code 1
           IFM_Module_Fence:I1.Data[56].7   // Port 4 Event Code 1
           IFM_Module_Fence:I1.Data[56].8   // Port 4 Event Code 2
           IFM_Module_Fence:I1.Data[56].9   // Port 4 Event Code 2
           IFM_Module_Fence:I1.Data[56].15   // Port 4 Event Code 2
           IFM_Module_Fence:I1.Data[57]   // Port 4 IO-Link Event Data
           IFM_Module_Fence:I1.Data[57].0   // Port 4 Event Instance
           IFM_Module_Fence:I1.Data[57].1   // Port 4 Event Instance
           IFM_Module_Fence:I1.Data[57].10   // Port 4 Event Code 1
           IFM_Module_Fence:I1.Data[57].11   // Port 4 Event Code 1
           IFM_Module_Fence:I1.Data[57].12   // Port 4 Event Code 1
           IFM_Module_Fence:I1.Data[57].13   // Port 4 Event Code 1
           IFM_Module_Fence:I1.Data[57].14   // Port 4 Event Code 1
           IFM_Module_Fence:I1.Data[57].15   // Port 4 Event Code 1
           IFM_Module_Fence:I1.Data[57].3   // Port 4 Event Source
           IFM_Module_Fence:I1.Data[50]   // Port 4 IO Link Status
           IFM_Module_Fence:I1.Data[54].4   // Port 4 Event Type
           IFM_Module_Fence:I1.Data[54].5   // Port 4 Event Type
           IFM_Module_Fence:I1.Data[54].6   // Port 4 Event Mode
           IFM_Module_Fence:I1.Data[57].8   // Port 4 Event Code 1
           IFM_Module_Fence:I1.Data[57].9   // Port 4 Event Code 1
           IFM_Module_Fence:I1.Data[57].2   // Port 4 Event Instance
           IFM_Module_Fence:I1.Data[58].0   // Port 4 Event Code 2
           IFM_Module_Fence:I1.Data[58].1   // Port 4 Event Code 2
           IFM_Module_Fence:I1.Data[58].10   // Reserved
           IFM_Module_Fence:I1.Data[58].11   // Reserved
           IFM_Module_Fence:I1.Data[58].12   // Reserved
           IFM_Module_Fence:I1.Data[58].13   // Reserved
           IFM_Module_Fence:I1.Data[58].14   // Reserved
           IFM_Module_Fence:I1.Data[58].15   // Reserved
           IFM_Module_Fence:I1.Data[58].2   // Port 4 Event Code 2
           IFM_Module_Fence:I1.Data[58].3   // Port 4 Event Code 2
           IFM_Module_Fence:I1.Data[58].4   // Port 4 Event Code 2
           IFM_Module_Fence:I1.Data[58].5   // Port 4 Event Code 2
           IFM_Module_Fence:I1.Data[58].6   // Port 4 Event Code 2
           IFM_Module_Fence:I1.Data[58].7   // Port 4 Event Code 2
           IFM_Module_Fence:I1.Data[58].8   // Reserved
           IFM_Module_Fence:I1.Data[58].9   // Reserved
           IFM_Module_Fence:I1.Data[58]   // Port 4 IO-Link Event Data
           IFM_Module_Fence:I1.Data[5]   // Read/Write Command Code; HandShake; Command Result
           IFM_Module_Fence:I1.Data[5].0   // TRUE if Read Acyclic Command Response
           IFM_Module_Fence:I1.Data[5].1   // TRUE if Write Acyclic Command Response
           IFM_Module_Fence:I1.Data[5].10   // Target Mode
           IFM_Module_Fence:I1.Data[5].11   // Target Mode
           IFM_Module_Fence:I1.Data[5].12   // Target Mode
           IFM_Module_Fence:I1.Data[5].13   // Target Mode
           IFM_Module_Fence:I1.Data[5].14   // Target Mode
           IFM_Module_Fence:I1.Data[5].15   // Target Mode
           IFM_Module_Fence:I1.Data[5].2   // Reserved
           IFM_Module_Fence:I1.Data[5].3   // Reserved
           IFM_Module_Fence:I1.Data[5].4   // Reserved
           IFM_Module_Fence:I1.Data[5].5   // Reserved
           IFM_Module_Fence:I1.Data[5].6   // Reserved
           IFM_Module_Fence:I1.Data[5].7   // TRUE if HandShake Response To Acyclic Command
           IFM_Module_Fence:I1.Data[5].8   // Target Mode
           IFM_Module_Fence:I1.Data[5].9   // Target Mode
           IFM_Module_Fence:I1.Data[59]   // Port 1 Input Process Data
           IFM_Module_Fence:I1.Data[60]   // Port 1 Input Process Data
           IFM_Module_Fence:I1.Data[61]   // Port 1 Input Process Data
           IFM_Module_Fence:I1.Data[62]   // Port 1 Input Process Data
           IFM_Module_Fence:I1.Data[63]   // Port 1 Input Process Data
           IFM_Module_Fence:I1.Data[64]   // Port 1 Input Process Data
           IFM_Module_Fence:I1.Data[65]   // Port 1 Input Process Data
           IFM_Module_Fence:I1.Data[66]   // Port 1 Input Process Data
           IFM_Module_Fence:I1.Data[67]   // Port 1 Input Process Data
           IFM_Module_Fence:I1.Data[68]   // Port 1 Input Process Data
           IFM_Module_Fence:I1.Data[6]   // Command Response Byte Length & Command Response or Diagnostic Data 0
           IFM_Module_Fence:I1.Data[6].0   // Command Byte Length Bit 0
           IFM_Module_Fence:I1.Data[6].1   // Command Byte Length Bit 1
           IFM_Module_Fence:I1.Data[6].10   // Command Response or Diagnostic Data 0
           IFM_Module_Fence:I1.Data[6].11   // Command Response or Diagnostic Data 0
           IFM_Module_Fence:I1.Data[6].12   // Command Response or Diagnostic Data 0
           IFM_Module_Fence:I1.Data[6].13   // Command Response or Diagnostic Data 0
           IFM_Module_Fence:I1.Data[6].14   // Command Response or Diagnostic Data 0
           IFM_Module_Fence:I1.Data[6].15   // Command Response or Diagnostic Data 0
           IFM_Module_Fence:I1.Data[6].2   // Command Byte Length Bit 2
           IFM_Module_Fence:I1.Data[6].3   // Command Byte Length Bit 3
           IFM_Module_Fence:I1.Data[6].4   // Command Byte Length Bit 4
           IFM_Module_Fence:I1.Data[6].5   // Command Byte Length Bit 5
           IFM_Module_Fence:I1.Data[6].6   // Command Byte Length Bit 6
           IFM_Module_Fence:I1.Data[6].7   // Command Byte Length Bit 7
           IFM_Module_Fence:I1.Data[6].8   // Command Response or Diagnostic Data 0
           IFM_Module_Fence:I1.Data[6].9   // Command Response or Diagnostic Data 0
           IFM_Module_Fence:I1.Data[69]   // Port 1 Input Process Data
           IFM_Module_Fence:I1.Data[70]   // Port 1 Input Process Data
           IFM_Module_Fence:I1.Data[71]   // Port 1 Input Process Data
           IFM_Module_Fence:I1.Data[72]   // Port 1 Input Process Data
           IFM_Module_Fence:I1.Data[73]   // Port 1 Input Process Data
           IFM_Module_Fence:I1.Data[74]   // Port 1 Input Process Data
           IFM_Module_Fence:I1.Data[75]   // Port 2 Input Process Data
           IFM_Module_Fence:I1.Data[76]   // Port 2 Input Process Data
           IFM_Module_Fence:I1.Data[77]   // Port 2 Input Process Data
           IFM_Module_Fence:I1.Data[78]   // Port 2 Input Process Data
           IFM_Module_Fence:I1.Data[7]   // Command Response Or Diagnostic Data 1
           IFM_Module_Fence:I1.Data[79]   // Port 2 Input Process Data
           IFM_Module_Fence:I1.Data[80]   // Port 2 Input Process Data
           IFM_Module_Fence:I1.Data[81]   // Port 2 Input Process Data
           IFM_Module_Fence:I1.Data[82]   // Port 2 Input Process Data
           IFM_Module_Fence:I1.Data[83]   // Port 2 Input Process Data
           IFM_Module_Fence:I1.Data[84]   // Port 2 Input Process Data
           IFM_Module_Fence:I1.Data[85]   // Port 2 Input Process Data
           IFM_Module_Fence:I1.Data[86]   // Port 2 Input Process Data
           IFM_Module_Fence:I1.Data[87]   // Port 2 Input Process Data
           IFM_Module_Fence:I1.Data[88]   // Port 2 Input Process Data
           IFM_Module_Fence:I1.Data[8]   // Command Response Or Diagnostic Data 3
           IFM_Module_Fence:I1.Data[89]   // Port 2 Input Process Data
           IFM_Module_Fence:I1.Data[90]   // Port 2 Input Process Data
           IFM_Module_Fence:I1.Data[91]   // Port 3 Input Process Data
           IFM_Module_Fence:I1.Data[92]   // Port 3 Input Process Data
           IFM_Module_Fence:I1.Data[93]   // Port 3 Input Process Data
           IFM_Module_Fence:I1.Data[94]   // Port 3 Input Process Data
           IFM_Module_Fence:I1.Data[95]   // Port 3 Input Process Data
           IFM_Module_Fence:I1.Data[96]   // Port 3 Input Process Data
           IFM_Module_Fence:I1.Data[97]   // Port 3 Input Process Data
           IFM_Module_Fence:I1.Data[98]   // Port 3 Input Process Data
           IFM_Module_Fence:I1.Data[9]   // Command Response Or Diagnostic Data 5
           IFM_Module_Fence:I1.Data[55]   // Port 4 IO-Link Event Data
           IFM_Module_Fence:I1.Data[54].7   // Port 4 Event Mode
           IFM_Module_Fence:I1.Data[57].4   // Port 4 Event Type
           IFM_Module_Fence:I1.Data[57].5   // Port 4 Event Type
           IFM_Module_Fence:I1.Data[57].6   // Port 4 Event Mode
           IFM_Module_Fence:I1.Data[57].7   // Port 4 Event Mode
           IFM_Module_Fence:I1.Data[99]   // Port 3 Input Process Data
           IFM_Module_Fence:I1.Data[50].4   // Port 4 IO-Link Data String Error
           IFM_Module_Fence:O1.Data[0].0   // Port 1 Pin 4 Digital Output
           IFM_Module_Fence:O1.Data[0].1   // Port 2 Pin 4 Digital Output
           IFM_Module_Fence:O1.Data[0].10   // Reserved
           IFM_Module_Fence:O1.Data[0].11   // Reserved
           IFM_Module_Fence:O1.Data[0].12   // Reserved
           IFM_Module_Fence:O1.Data[0].13   // Reserved
           IFM_Module_Fence:O1.Data[0].14   // Reserved
           IFM_Module_Fence:O1.Data[0].15   // Reserved
           IFM_Module_Fence:O1.Data[0].2   // Port 3 Pin 4 Digital Output
           IFM_Module_Fence:O1.Data[0].3   // Port 4 Pin 4 Digital Output
           IFM_Module_Fence:O1.Data[0].4   // Reserved
           IFM_Module_Fence:O1.Data[0].5   // Reserved
           IFM_Module_Fence:O1.Data[0].6   // Reserved
           IFM_Module_Fence:O1.Data[0].7   // Reserved
           IFM_Module_Fence:O1.Data[0].8   // Reserved
           IFM_Module_Fence:O1.Data[0].9   // Reserved
           IFM_Module_Fence:O1.Data[10]   // Command Data Array 8
           IFM_Module_Fence:O1.Data[11]   // Command Data Array 10
           IFM_Module_Fence:O1.Data[12]   // Command Data Array 12
           IFM_Module_Fence:O1.Data[13]   // Command Data Array 14
           IFM_Module_Fence:O1.Data[14]   // Command Data Array 16
           IFM_Module_Fence:O1.Data[1]   // Reserved
           IFM_Module_Fence:O1.Data[15]   // Command Data Array 18
           IFM_Module_Fence:O1.Data[16]   // Command Data Array 20
           IFM_Module_Fence:O1.Data[22]   // Reserved
           IFM_Module_Fence:O1.Data[23]   // Port 1 Digital Output Process Data
           IFM_Module_Fence:O1.Data[24]   // Port 1 Digital Output Process Data
           IFM_Module_Fence:O1.Data[25]   // Port 1 Digital Output Process Data
           IFM_Module_Fence:O1.Data[26]   // Port 1 Digital Output Process Data
           IFM_Module_Fence:O1.Data[27]   // Port 1 Digital Output Process Data
           IFM_Module_Fence:O1.Data[28]   // Port 1 Digital Output Process Data
           IFM_Module_Fence:O1.Data[29]   // Port 1 Digital Output Process Data
           IFM_Module_Fence:O1.Data[2]   // AL1x2x Port Number
           IFM_Module_Fence:O1.Data[30]   // Port 1 Digital Output Process Data
           IFM_Module_Fence:O1.Data[31]   // Port 1 Digital Output Process Data
           IFM_Module_Fence:O1.Data[32]   // Port 1 Digital Output Process Data
           IFM_Module_Fence:O1.Data[33]   // Port 1 Digital Output Process Data
           IFM_Module_Fence:O1.Data[34]   // Port 1 Digital Output Process Data
           IFM_Module_Fence:O1.Data[35]   // Port 1 Digital Output Process Data
           IFM_Module_Fence:O1.Data[36]   // Port 1 Digital Output Process Data
           IFM_Module_Fence:O1.Data[37]   // Port 1 Digital Output Process Data
           IFM_Module_Fence:O1.Data[38]   // Port 1 Digital Output Process Data
           IFM_Module_Fence:O1.Data[39]   // Port 2 Digital Output Process Data
           IFM_Module_Fence:O1.Data[3]   // Index Number
           IFM_Module_Fence:O1.Data[40]   // Port 2 Digital Output Process Data
           IFM_Module_Fence:O1.Data[41]   // Port 2 Digital Output Process Data
           IFM_Module_Fence:O1.Data[42]   // Port 2 Digital Output Process Data
           IFM_Module_Fence:O1.Data[43]   // Port 2 Digital Output Process Data
           IFM_Module_Fence:O1.Data[44]   // Port 2 Digital Output Process Data
           IFM_Module_Fence:O1.Data[45]   // Port 2 Digital Output Process Data
           IFM_Module_Fence:O1.Data[46]   // Port 2 Digital Output Process Data
           IFM_Module_Fence:O1.Data[47]   // Port 2 Digital Output Process Data
           IFM_Module_Fence:O1.Data[48]   // Port 2 Digital Output Process Data
           IFM_Module_Fence:O1.Data[49]   // Port 2 Digital Output Process Data
           IFM_Module_Fence:O1.Data[4]   // SubIndex Number
           IFM_Module_Fence:O1.Data[50]   // Port 2 Digital Output Process Data
           IFM_Module_Fence:O1.Data[51]   // Port 2 Digital Output Process Data
           IFM_Module_Fence:O1.Data[52]   // Port 2 Digital Output Process Data
           IFM_Module_Fence:O1.Data[53]   // Port 2 Digital Output Process Data
           IFM_Module_Fence:O1.Data[54]   // Port 2 Digital Output Process Data
           IFM_Module_Fence:O1.Data[55]   // Port 3 Digital Output Process Data
           IFM_Module_Fence:O1.Data[56]   // Port 3 Digital Output Process Data
           IFM_Module_Fence:O1.Data[57]   // Port 3 Digital Output Process Data
           IFM_Module_Fence:O1.Data[58]   // Port 3 Digital Output Process Data
           IFM_Module_Fence:O1.Data[59]   // Port 3 Digital Output Process Data
           IFM_Module_Fence:O1.Data[5]   // Read/Write Command Code; Trigger Bit; Command Byte Length
           IFM_Module_Fence:O1.Data[5].0   // Set TRUE to Read
           IFM_Module_Fence:O1.Data[5].1   // Set TRUE to Write
           IFM_Module_Fence:O1.Data[5].10   // Command Byte Length Bit 2
           IFM_Module_Fence:O1.Data[5].11   // Command Byte Length Bit 3
           IFM_Module_Fence:O1.Data[5].12   // Command Byte Length Bit 4
           IFM_Module_Fence:O1.Data[5].13   // Command Byte Length Bit 5
           IFM_Module_Fence:O1.Data[5].14   // Command Byte Length Bit 6
           IFM_Module_Fence:O1.Data[5].15   // Command Byte Length Bit 7
           IFM_Module_Fence:O1.Data[5].2   // Reserved
           IFM_Module_Fence:O1.Data[5].3   // Reserved
           IFM_Module_Fence:O1.Data[5].4   // Reserved
           IFM_Module_Fence:O1.Data[5].5   // Reserved
           IFM_Module_Fence:O1.Data[5].6   // Reserved
           IFM_Module_Fence:O1.Data[5].8   // Command Byte Length Bit 0
           IFM_Module_Fence:O1.Data[5].9   // Command Byte Length Bit 1
           IFM_Module_Fence:O1.Data[60]   // Port 3 Digital Output Process Data
           IFM_Module_Fence:O1.Data[61]   // Port 3 Digital Output Process Data
           IFM_Module_Fence:O1.Data[62]   // Port 3 Digital Output Process Data
           IFM_Module_Fence:O1.Data[63]   // Port 3 Digital Output Process Data
           IFM_Module_Fence:O1.Data[64]   // Port 3 Digital Output Process Data
           IFM_Module_Fence:O1.Data[65]   // Port 3 Digital Output Process Data
           IFM_Module_Fence:O1.Data[66]   // Port 3 Digital Output Process Data
           IFM_Module_Fence:O1.Data[67]   // Port 3 Digital Output Process Data
           IFM_Module_Fence:O1.Data[68]   // Port 3 Digital Output Process Data
           IFM_Module_Fence:O1.Data[69]   // Port 3 Digital Output Process Data
           IFM_Module_Fence:O1.Data[6]   // Command Data Array 0
           IFM_Module_Fence:O1.Data[70]   // Port 3 Digital Output Process Data
           IFM_Module_Fence:O1.Data[71]   // Port 4 Digital Output Process Data
           IFM_Module_Fence:O1.Data[72]   // Port 4 Digital Output Process Data
           IFM_Module_Fence:O1.Data[73]   // Port 4 Digital Output Process Data
           IFM_Module_Fence:O1.Data[74]   // Port 4 Digital Output Process Data
           IFM_Module_Fence:O1.Data[75]   // Port 4 Digital Output Process Data
           IFM_Module_Fence:O1.Data[76]   // Port 4 Digital Output Process Data
           IFM_Module_Fence:O1.Data[77]   // Port 4 Digital Output Process Data
           IFM_Module_Fence:O1.Data[78]   // Port 4 Digital Output Process Data
           IFM_Module_Fence:O1.Data[79]   // Port 4 Digital Output Process Data
           IFM_Module_Fence:O1.Data[7]   // Command Data Array 2
           IFM_Module_Fence:O1.Data[80]   // Port 4 Digital Output Process Data
           IFM_Module_Fence:O1.Data[81]   // Port 4 Digital Output Process Data
           IFM_Module_Fence:O1.Data[82]   // Port 4 Digital Output Process Data
           IFM_Module_Fence:O1.Data[83]   // Port 4 Digital Output Process Data
           IFM_Module_Fence:O1.Data[84]   // Port 4 Digital Output Process Data
           IFM_Module_Fence:O1.Data[85]   // Port 4 Digital Output Process Data
           IFM_Module_Fence:O1.Data[86]   // Port 4 Digital Output Process Data
           IFM_Module_Fence:O1.Data[8]   // Command Data Array 4
           IFM_Module_Fence:O1.Data[9]   // Command Data Array 6
           IFM_Module_Fence:O1.Data[5].7   // Trigger Acyclic Command
           IFM_Module_Fence:O1.Data[17]   // Command Data Array 22
           IFM_Module_Fence:O1.Data[18]   // Command Data Array 24
           IFM_Module_Fence:O1.Data[19]   // Command Data Array 26
           IFM_Module_Fence:O1.Data[20]   // Command Data Array 28
           IFM_Module_Fence:O1.Data[21]   // Command Data Array 30
           IFM_Module_Fence:O1.Data[0]   // AL1x2x Digital Output Status
      IFM_Module_RobotArm : vendor 322 type 12 code 1120 (Ethernet 192.168.1.42, rev 1.5, StandardDataDriven RPI 10 ms)
           IFM_Module_RobotArm:I1.Data[10]   // Command Response Or Diagnostic Data 7
           IFM_Module_RobotArm:I1.Data[0].0   // Port 1 Pin 4
           IFM_Module_RobotArm:I1.Data[0].1   // Port 2 Pin 4
           IFM_Module_RobotArm:I1.Data[0].10   // Port 3 Pin 2
           IFM_Module_RobotArm:I1.Data[0].11   // Port 4 Pin 2
           IFM_Module_RobotArm:I1.Data[0].12   // Reserved
           IFM_Module_RobotArm:I1.Data[0].13   // Reserved
           IFM_Module_RobotArm:I1.Data[0].14   // Reserved
           IFM_Module_RobotArm:I1.Data[0].15   // Reserved
           IFM_Module_RobotArm:I1.Data[0].2   // Port 3 Pin 4
           IFM_Module_RobotArm:I1.Data[0].3   // Port 4 Pin 4
           IFM_Module_RobotArm:I1.Data[0].4   // Reserved
           IFM_Module_RobotArm:I1.Data[0].5   // Reserved
           IFM_Module_RobotArm:I1.Data[0].6   // Reserved
           IFM_Module_RobotArm:I1.Data[0].7   // Reserved
           IFM_Module_RobotArm:I1.Data[0].8   // Port 1 Pin 2
           IFM_Module_RobotArm:I1.Data[0].9   // Port 2 Pin 2
           IFM_Module_RobotArm:I1.Data[100]   // Port 3 Input Process Data
           IFM_Module_RobotArm:I1.Data[101]   // Port 3 Input Process Data
           IFM_Module_RobotArm:I1.Data[102]   // Port 3 Input Process Data
           IFM_Module_RobotArm:I1.Data[103]   // Port 3 Input Process Data
           IFM_Module_RobotArm:I1.Data[104]   // Port 3 Input Process Data
           IFM_Module_RobotArm:I1.Data[105]   // Port 3 Input Process Data
           IFM_Module_RobotArm:I1.Data[106]   // Port 3 Input Process Data
           IFM_Module_RobotArm:I1.Data[107]   // Port 4 Input Process Data
           IFM_Module_RobotArm:I1.Data[108]   // Port 4 Input Process Data
           IFM_Module_RobotArm:I1.Data[109]   // Port 4 Input Process Data
           IFM_Module_RobotArm:I1.Data[11]   // Command Response Or Diagnostic Data 9
           IFM_Module_RobotArm:I1.Data[110]   // Port 4 Input Process Data
           IFM_Module_RobotArm:I1.Data[111]   // Port 4 Input Process Data
           IFM_Module_RobotArm:I1.Data[112]   // Port 4 Input Process Data
           IFM_Module_RobotArm:I1.Data[113]   // Port 4 Input Process Data
           IFM_Module_RobotArm:I1.Data[114]   // Port 4 Input Process Data
           IFM_Module_RobotArm:I1.Data[115]   // Port 4 Input Process Data
           IFM_Module_RobotArm:I1.Data[116]   // Port 4 Input Process Data
           IFM_Module_RobotArm:I1.Data[117]   // Port 4 Input Process Data
           IFM_Module_RobotArm:I1.Data[118]   // Port 4 Input Process Data
           IFM_Module_RobotArm:I1.Data[119]   // Port 4 Input Process Data
           IFM_Module_RobotArm:I1.Data[7]   // Command Response Or Diagnostic Data 1
           IFM_Module_RobotArm:I1.Data[120]   // Port 4 Input Process Data
           IFM_Module_RobotArm:I1.Data[121]   // Port 4 Input Process Data
           IFM_Module_RobotArm:I1.Data[122]   // Port 4 Input Process Data
           IFM_Module_RobotArm:I1.Data[12]   // Command Response Or Diagnostic Data 11
           IFM_Module_RobotArm:I1.Data[13]   // Command Response Or Diagnostic Data 13
           IFM_Module_RobotArm:I1.Data[14]   // Command Response Or Diagnostic Data 15
           IFM_Module_RobotArm:I1.Data[15]   // Command Response Or Diagnostic Data 17
           IFM_Module_RobotArm:I1.Data[16]   // Command Response Or Diagnostic Data 19
           IFM_Module_RobotArm:I1.Data[17]   // Command Response Or Diagnostic Data 21
           IFM_Module_RobotArm:I1.Data[18]   // Command Response Or Diagnostic Data 23
           IFM_Module_RobotArm:I1.Data[1]   // AL1x2x Digital Input Short/Overload Status
           IFM_Module_RobotArm:I1.Data[1].0   // Port 1 Short/Overload
           IFM_Module_RobotArm:I1.Data[1].1   // Port 2 Short/Overload
           IFM_Module_RobotArm:I1.Data[1].10   // Reserved
           IFM_Module_RobotArm:I1.Data[1].11   // Reserved
           IFM_Module_RobotArm:I1.Data[1].12   // Reserved
           IFM_Module_RobotArm:I1.Data[1].13   // Reserved
           IFM_Module_RobotArm:I1.Data[1].14   // Reserved
           IFM_Module_RobotArm:I1.Data[1].15   // Reserved
           IFM_Module_RobotArm:I1.Data[1].2   // Port 3 Short/Overload
           IFM_Module_RobotArm:I1.Data[1].3   // Port 4 Short/Overload
           IFM_Module_RobotArm:I1.Data[1].4   // Reserved
           IFM_Module_RobotArm:I1.Data[1].5   // Reserved
           IFM_Module_RobotArm:I1.Data[1].6   // Reserved
           IFM_Module_RobotArm:I1.Data[1].7   // Reserved
           IFM_Module_RobotArm:I1.Data[1].8   // Reserved
           IFM_Module_RobotArm:I1.Data[1].9   // Reserved
           IFM_Module_RobotArm:I1.Data[19]   // Command Response Or Diagnostic Data 25
           IFM_Module_RobotArm:I1.Data[20]   // Command Response Or Diagnostic Data 27
           IFM_Module_RobotArm:I1.Data[21]   // Command Response Or Diagnostic Data 29
           IFM_Module_RobotArm:I1.Data[23].0   // Port 1 IO-Link Mode
           IFM_Module_RobotArm:I1.Data[22]   // Command Response Or Diagnostic Data 31
           IFM_Module_RobotArm:I1.Data[23].10   // Reserved
           IFM_Module_RobotArm:I1.Data[23].11   // Reserved
           IFM_Module_RobotArm:I1.Data[23].12   // Reserved
           IFM_Module_RobotArm:I1.Data[23].13   // Reserved
           IFM_Module_RobotArm:I1.Data[23].14   // Reserved
           IFM_Module_RobotArm:I1.Data[23].15   // Reserved
           IFM_Module_RobotArm:I1.Data[23].2   // Port 1 IO-Link Data Invalid
           IFM_Module_RobotArm:I1.Data[23].3   // Port 1 Incorrect Vendor or Device ID
           IFM_Module_RobotArm:I1.Data[23].5   // Reserved
           IFM_Module_RobotArm:I1.Data[23].6   // Reserved
           IFM_Module_RobotArm:I1.Data[23].7   // Reserved
           IFM_Module_RobotArm:I1.Data[23].8   // Reserved
           IFM_Module_RobotArm:I1.Data[23].9   // Reserved
           IFM_Module_RobotArm:I1.Data[24]   // Port 1 Vendor ID
           IFM_Module_RobotArm:I1.Data[25]   // Port 1 Device ID (Low Word)
           IFM_Module_RobotArm:I1.Data[26]   // Port 1 Device ID (High Word)
           IFM_Module_RobotArm:I1.Data[0]   // AL1x2x Digital Input Status
           IFM_Module_RobotArm:I1.Data[27]   // Port 1 IO-Link Event Data
           IFM_Module_RobotArm:I1.Data[27].0   // Port 1 Event Instance
           IFM_Module_RobotArm:I1.Data[27].1   // Port 1 Event Instance
           IFM_Module_RobotArm:I1.Data[27].10   // Port 1 Event Code 1
           IFM_Module_RobotArm:I1.Data[27].11   // Port 1 Event Code 1
           IFM_Module_RobotArm:I1.Data[27].12   // Port 1 Event Code 1
           IFM_Module_RobotArm:I1.Data[27].13   // Port 1 Event Code 1
           IFM_Module_RobotArm:I1.Data[27].14   // Port 1 Event Code 1
           IFM_Module_RobotArm:I1.Data[27].15   // Port 1 Event Code 1
           IFM_Module_RobotArm:I1.Data[27].3   // Port 1 Event Source
           IFM_Module_RobotArm:I1.Data[27].8   // Port 1 Event Code 1
           IFM_Module_RobotArm:I1.Data[27].9   // Port 1 Event Code 1
           IFM_Module_RobotArm:I1.Data[28].0   // Port 1 Event Code 2
           IFM_Module_RobotArm:I1.Data[28].1   // Port 1 Event Code 2
           IFM_Module_RobotArm:I1.Data[28].10   // Port 1 Event Instance
           IFM_Module_RobotArm:I1.Data[27].2   // Port 1 Event Instance
           IFM_Module_RobotArm:I1.Data[28].12   // Port 1 Event Type
           IFM_Module_RobotArm:I1.Data[28].13   // Port 1 Event Type
           IFM_Module_RobotArm:I1.Data[28].14   // Port 1 Event Mode
           IFM_Module_RobotArm:I1.Data[28].15   // Port 1 Event Mode
           IFM_Module_RobotArm:I1.Data[28].2   // Port 1 Event Code 2
           IFM_Module_RobotArm:I1.Data[28].3   // Port 1 Event Code 2
           IFM_Module_RobotArm:I1.Data[28].4   // Port 1 Event Code 2
           IFM_Module_RobotArm:I1.Data[28].5   // Port 1 Event Code 2
           IFM_Module_RobotArm:I1.Data[28].6   // Port 1 Event Code 2
           IFM_Module_RobotArm:I1.Data[28].7   // Port 1 Event Code 2
           IFM_Module_RobotArm:I1.Data[28].11   // Port 1 Event Source
           IFM_Module_RobotArm:I1.Data[28].8   // Port 1 Event Instance
           IFM_Module_RobotArm:I1.Data[28].9   // Port 1 Event Instance
           IFM_Module_RobotArm:I1.Data[29].0   // Port 1 Event Code 1
           IFM_Module_RobotArm:I1.Data[29].1   // Port 1 Event Code 1
           IFM_Module_RobotArm:I1.Data[29]   // Port 1 IO-Link Event Data
           IFM_Module_RobotArm:I1.Data[29].10   // Port 1 Event Code 2
           IFM_Module_RobotArm:I1.Data[29].11   // Port 1 Event Code 2
           IFM_Module_RobotArm:I1.Data[29].12   // Port 1 Event Code 2
           IFM_Module_RobotArm:I1.Data[29].13   // Port 1 Event Code 2
           IFM_Module_RobotArm:I1.Data[29].14   // Port 1 Event Code 2
           IFM_Module_RobotArm:I1.Data[29].2   // Port 1 Event Code 1
           IFM_Module_RobotArm:I1.Data[29].3   // Port 1 Event Code 1
           IFM_Module_RobotArm:I1.Data[29].4   // Port 1 Event Code 1
           IFM_Module_RobotArm:I1.Data[29].5   // Port 1 Event Code 1
           IFM_Module_RobotArm:I1.Data[29].6   // Port 1 Event Code 1
           IFM_Module_RobotArm:I1.Data[29].7   // Port 1 Event Code 1
           IFM_Module_RobotArm:I1.Data[29].8   // Port 1 Event Code 2
           IFM_Module_RobotArm:I1.Data[29].9   // Port 1 Event Code 2
           IFM_Module_RobotArm:I1.Data[2]   // Port Number
           IFM_Module_RobotArm:I1.Data[29].15   // Port 1 Event Code 2
           IFM_Module_RobotArm:I1.Data[30]   // Port 1 IO-Link Event Data
           IFM_Module_RobotArm:I1.Data[30].0   // Port 1 Event Instance
           IFM_Module_RobotArm:I1.Data[30].1   // Port 1 Event Instance
           IFM_Module_RobotArm:I1.Data[30].10   // Port 1 Event Code 1
           IFM_Module_RobotArm:I1.Data[30].11   // Port 1 Event Code 1
           IFM_Module_RobotArm:I1.Data[30].12   // Port 1 Event Code 1
           IFM_Module_RobotArm:I1.Data[30].13   // Port 1 Event Code 1
           IFM_Module_RobotArm:I1.Data[30].14   // Port 1 Event Code 1
           IFM_Module_RobotArm:I1.Data[30].15   // Port 1 Event Code 1
           IFM_Module_RobotArm:I1.Data[30].3   // Port 1 Event Source
           IFM_Module_RobotArm:I1.Data[23]   // Port 1 IO Link Status
           IFM_Module_RobotArm:I1.Data[27].4   // Port 1 Event Type
           IFM_Module_RobotArm:I1.Data[27].5   // Port 1 Event Type
           IFM_Module_RobotArm:I1.Data[27].6   // Port 1 Event Mode
           IFM_Module_RobotArm:I1.Data[30].8   // Port 1 Event Code 1
           IFM_Module_RobotArm:I1.Data[30].9   // Port 1 Event Code 1
           IFM_Module_RobotArm:I1.Data[30].2   // Port 1 Event Instance
           IFM_Module_RobotArm:I1.Data[31].0   // Port 1 Event Code 2
           IFM_Module_RobotArm:I1.Data[31].1   // Port 1 Event Code 2
           IFM_Module_RobotArm:I1.Data[31].10   // Reserved
           IFM_Module_RobotArm:I1.Data[31].11   // Reserved
           IFM_Module_RobotArm:I1.Data[31].12   // Reserved
           IFM_Module_RobotArm:I1.Data[31].13   // Reserved
           IFM_Module_RobotArm:I1.Data[31].14   // Reserved
           IFM_Module_RobotArm:I1.Data[31].15   // Reserved
           IFM_Module_RobotArm:I1.Data[31].2   // Port 1 Event Code 2
           IFM_Module_RobotArm:I1.Data[31].3   // Port 1 Event Code 2
           IFM_Module_RobotArm:I1.Data[31].4   // Port 1 Event Code 2
           IFM_Module_RobotArm:I1.Data[31].5   // Port 1 Event Code 2
           IFM_Module_RobotArm:I1.Data[31].6   // Port 1 Event Code 2
           IFM_Module_RobotArm:I1.Data[31].7   // Port 1 Event Code 2
           IFM_Module_RobotArm:I1.Data[31].8   // Reserved
           IFM_Module_RobotArm:I1.Data[31].9   // Reserved
           IFM_Module_RobotArm:I1.Data[27].7   // Port 1 Event Mode
           IFM_Module_RobotArm:I1.Data[32].0   // Port 2 IO-Link Mode
           IFM_Module_RobotArm:I1.Data[23].1   // Port 1 NO IO-Link Device Connected
           IFM_Module_RobotArm:I1.Data[32].10   // Reserved
           IFM_Module_RobotArm:I1.Data[32].11   // Reserved
           IFM_Module_RobotArm:I1.Data[32].12   // Reserved
           IFM_Module_RobotArm:I1.Data[32].13   // Reserved
           IFM_Module_RobotArm:I1.Data[32].14   // Reserved
           IFM_Module_RobotArm:I1.Data[32].15   // Reserved
           IFM_Module_RobotArm:I1.Data[32].2   // Port 2 IO-Link Data Invalid
           IFM_Module_RobotArm:I1.Data[32].3   // Port 2 Incorrect Vendor or Device ID
           IFM_Module_RobotArm:I1.Data[23].4   // Port 1 IO-Link Data String Error
           IFM_Module_RobotArm:I1.Data[32].5   // Reserved
           IFM_Module_RobotArm:I1.Data[32].6   // Reserved
           IFM_Module_RobotArm:I1.Data[32].7   // Reserved
           IFM_Module_RobotArm:I1.Data[32].8   // Reserved
           IFM_Module_RobotArm:I1.Data[32].9   // Reserved
           IFM_Module_RobotArm:I1.Data[33]   // Port 2 Vendor ID
           IFM_Module_RobotArm:I1.Data[34]   // Port 2 Device ID (Low Word)
           IFM_Module_RobotArm:I1.Data[35]   // Port 2 Device ID (High Word)
           IFM_Module_RobotArm:I1.Data[31]   // Port 1 IO-Link Event Data
           IFM_Module_RobotArm:I1.Data[36]   // Port 2 IO-Link Event Data
           IFM_Module_RobotArm:I1.Data[36].0   // Port 2 Event Instance
           IFM_Module_RobotArm:I1.Data[36].1   // Port 2 Event Instance
           IFM_Module_RobotArm:I1.Data[36].10   // Port 2 Event Code 1
           IFM_Module_RobotArm:I1.Data[36].11   // Port 2 Event Code 1
           IFM_Module_RobotArm:I1.Data[36].12   // Port 2 Event Code 1
           IFM_Module_RobotArm:I1.Data[36].13   // Port 2 Event Code 1
           IFM_Module_RobotArm:I1.Data[36].14   // Port 2 Event Code 1
           IFM_Module_RobotArm:I1.Data[36].15   // Port 2 Event Code 1
           IFM_Module_RobotArm:I1.Data[36].3   // Port 2 Event Source
           IFM_Module_RobotArm:I1.Data[30].4   // Port 1 Event Type
           IFM_Module_RobotArm:I1.Data[30].5   // Port 1 Event Type
           IFM_Module_RobotArm:I1.Data[30].6   // Port 1 Event Mode
           IFM_Module_RobotArm:I1.Data[30].7   // Port 1 Event Mode
           IFM_Module_RobotArm:I1.Data[36].8   // Port 2 Event Code 1
           IFM_Module_RobotArm:I1.Data[36].9   // Port 2 Event Code 1
           IFM_Module_RobotArm:I1.Data[28]   // Port 1 IO-Link Event Data
           IFM_Module_RobotArm:I1.Data[37].0   // Port 2 Event Code 2
           IFM_Module_RobotArm:I1.Data[37].1   // Port 2 Event Code 2
           IFM_Module_RobotArm:I1.Data[37].10   // Port 2 Event Instance
           IFM_Module_RobotArm:I1.Data[36].2   // Port 2 Event Instance
           IFM_Module_RobotArm:I1.Data[37].12   // Port 2 Event Type
           IFM_Module_RobotArm:I1.Data[37].13   // Port 2 Event Type
           IFM_Module_RobotArm:I1.Data[37].14   // Port 2 Event Mode
           IFM_Module_RobotArm:I1.Data[37].15   // Port 2 Event Mode
           IFM_Module_RobotArm:I1.Data[37].2   // Port 2 Event Code 2
           IFM_Module_RobotArm:I1.Data[37].3   // Port 2 Event Code 2
           IFM_Module_RobotArm:I1.Data[37].4   // Port 2 Event Code 2
           IFM_Module_RobotArm:I1.Data[37].5   // Port 2 Event Code 2
           IFM_Module_RobotArm:I1.Data[37].6   // Port 2 Event Code 2
           IFM_Module_RobotArm:I1.Data[37].7   // Port 2 Event Code 2
           IFM_Module_RobotArm:I1.Data[37].11   // Port 2 Event Source
           IFM_Module_RobotArm:I1.Data[37].8   // Port 2 Event Instance
           IFM_Module_RobotArm:I1.Data[37].9   // Port 2 Event Instance
           IFM_Module_RobotArm:I1.Data[38].0   // Port 2 Event Code 1
           IFM_Module_RobotArm:I1.Data[38].1   // Port 2 Event Code 1
           IFM_Module_RobotArm:I1.Data[38]   // Port 2 IO-Link Event Data
           IFM_Module_RobotArm:I1.Data[38].10   // Port 2 Event Code 2
           IFM_Module_RobotArm:I1.Data[38].11   // Port 2 Event Code 2
           IFM_Module_RobotArm:I1.Data[38].12   // Port 2 Event Code 2
           IFM_Module_RobotArm:I1.Data[38].13   // Port 2 Event Code 2
           IFM_Module_RobotArm:I1.Data[38].14   // Port 2 Event Code 2
           IFM_Module_RobotArm:I1.Data[38].2   // Port 2 Event Code 1
           IFM_Module_RobotArm:I1.Data[38].3   // Port 2 Event Code 1
           IFM_Module_RobotArm:I1.Data[38].4   // Port 2 Event Code 1
           IFM_Module_RobotArm:I1.Data[38].5   // Port 2 Event Code 1
           IFM_Module_RobotArm:I1.Data[38].6   // Port 2 Event Code 1
           IFM_Module_RobotArm:I1.Data[38].7   // Port 2 Event Code 1
           IFM_Module_RobotArm:I1.Data[38].8   // Port 2 Event Code 2
           IFM_Module_RobotArm:I1.Data[38].9   // Port 2 Event Code 2
           IFM_Module_RobotArm:I1.Data[38].15   // Port 2 Event Code 2
           IFM_Module_RobotArm:I1.Data[39]   // Port 2 IO-Link Event Data
           IFM_Module_RobotArm:I1.Data[39].0   // Port 2 Event Instance
           IFM_Module_RobotArm:I1.Data[39].1   // Port 2 Event Instance
           IFM_Module_RobotArm:I1.Data[39].10   // Port 2 Event Code 1
           IFM_Module_RobotArm:I1.Data[39].11   // Port 2 Event Code 1
           IFM_Module_RobotArm:I1.Data[39].12   // Port 2 Event Code 1
           IFM_Module_RobotArm:I1.Data[39].13   // Port 2 Event Code 1
           IFM_Module_RobotArm:I1.Data[39].14   // Port 2 Event Code 1
           IFM_Module_RobotArm:I1.Data[39].15   // Port 2 Event Code 1
           IFM_Module_RobotArm:I1.Data[39].3   // Port 2 Event Source
           IFM_Module_RobotArm:I1.Data[32]   // Port 2 IO Link Status
           IFM_Module_RobotArm:I1.Data[36].4   // Port 2 Event Type
           IFM_Module_RobotArm:I1.Data[36].5   // Port 2 Event Type
           IFM_Module_RobotArm:I1.Data[36].6   // Port 2 Event Mode
           IFM_Module_RobotArm:I1.Data[39].8   // Port 2 Event Code 1
           IFM_Module_RobotArm:I1.Data[39].9   // Port 2 Event Code 1
           IFM_Module_RobotArm:I1.Data[3]   // Index Number
           IFM_Module_RobotArm:I1.Data[39].2   // Port 2 Event Instance
           IFM_Module_RobotArm:I1.Data[40].0   // Port 2 Event Code 2
           IFM_Module_RobotArm:I1.Data[40].1   // Port 2 Event Code 2
           IFM_Module_RobotArm:I1.Data[40].10   // Reserved
           IFM_Module_RobotArm:I1.Data[40].11   // Reserved
           IFM_Module_RobotArm:I1.Data[40].12   // Reserved
           IFM_Module_RobotArm:I1.Data[40].13   // Reserved
           IFM_Module_RobotArm:I1.Data[40].14   // Reserved
           IFM_Module_RobotArm:I1.Data[40].15   // Reserved
           IFM_Module_RobotArm:I1.Data[40].2   // Port 2 Event Code 2
           IFM_Module_RobotArm:I1.Data[40].3   // Port 2 Event Code 2
           IFM_Module_RobotArm:I1.Data[40].4   // Port 2 Event Code 2
           IFM_Module_RobotArm:I1.Data[40].5   // Port 2 Event Code 2
           IFM_Module_RobotArm:I1.Data[40].6   // Port 2 Event Code 2
           IFM_Module_RobotArm:I1.Data[40].7   // Port 2 Event Code 2
           IFM_Module_RobotArm:I1.Data[40].8   // Reserved
           IFM_Module_RobotArm:I1.Data[40].9   // Reserved
           IFM_Module_RobotArm:I1.Data[36].7   // Port 2 Event Mode
           IFM_Module_RobotArm:I1.Data[41].0   // Port 3 IO-Link Mode
           IFM_Module_RobotArm:I1.Data[32].1   // Port 2 NO IO-Link Device Connected
           IFM_Module_RobotArm:I1.Data[41].10   // Reserved
           IFM_Module_RobotArm:I1.Data[41].11   // Reserved
           IFM_Module_RobotArm:I1.Data[41].12   // Reserved
           IFM_Module_RobotArm:I1.Data[41].13   // Reserved
           IFM_Module_RobotArm:I1.Data[41].14   // Reserved
           IFM_Module_RobotArm:I1.Data[41].15   // Reserved
           IFM_Module_RobotArm:I1.Data[41].2   // Port 3 IO-Link Data Invalid
           IFM_Module_RobotArm:I1.Data[41].3   // Port 3 Incorrect Vendor or Device ID
           IFM_Module_RobotArm:I1.Data[32].4   // Port 2 IO-Link Data String Error
           IFM_Module_RobotArm:I1.Data[41].5   // Reserved
           IFM_Module_RobotArm:I1.Data[41].6   // Reserved
           IFM_Module_RobotArm:I1.Data[41].7   // Reserved
           IFM_Module_RobotArm:I1.Data[41].8   // Reserved
           IFM_Module_RobotArm:I1.Data[41].9   // Reserved
           IFM_Module_RobotArm:I1.Data[42]   // Port 3 Vendor ID
           IFM_Module_RobotArm:I1.Data[43]   // Port 3 Device ID (Low Word)
           IFM_Module_RobotArm:I1.Data[44]   // Port 3 Device ID (High Word)
           IFM_Module_RobotArm:I1.Data[40]   // Port 2 IO-Link Event Data
           IFM_Module_RobotArm:I1.Data[45]   // Port 3 IO-Link Event Data
           IFM_Module_RobotArm:I1.Data[45].0   // Port 3 Event Instance
           IFM_Module_RobotArm:I1.Data[45].1   // Port 3 Event Instance
           IFM_Module_RobotArm:I1.Data[45].10   // Port 3 Event Code 1
           IFM_Module_RobotArm:I1.Data[45].11   // Port 3 Event Code 1
           IFM_Module_RobotArm:I1.Data[45].12   // Port 3 Event Code 1
           IFM_Module_RobotArm:I1.Data[45].13   // Port 3 Event Code 1
           IFM_Module_RobotArm:I1.Data[45].14   // Port 3 Event Code 1
           IFM_Module_RobotArm:I1.Data[45].15   // Port 3 Event Code 1
           IFM_Module_RobotArm:I1.Data[45].3   // Port 3 Event Source
           IFM_Module_RobotArm:I1.Data[39].4   // Port 2 Event Type
           IFM_Module_RobotArm:I1.Data[39].5   // Port 2 Event Type
           IFM_Module_RobotArm:I1.Data[39].6   // Port 2 Event Mode
           IFM_Module_RobotArm:I1.Data[39].7   // Port 2 Event Mode
           IFM_Module_RobotArm:I1.Data[45].8   // Port 3 Event Code 1
           IFM_Module_RobotArm:I1.Data[45].9   // Port 3 Event Code 1
           IFM_Module_RobotArm:I1.Data[37]   // Port 2 IO-Link Event Data
           IFM_Module_RobotArm:I1.Data[46].0   // Port 3 Event Code 2
           IFM_Module_RobotArm:I1.Data[46].1   // Port 3 Event Code 2
           IFM_Module_RobotArm:I1.Data[46].10   // Port 3 Event Instance
           IFM_Module_RobotArm:I1.Data[45].2   // Port 3 Event Instance
           IFM_Module_RobotArm:I1.Data[46].12   // Port 3 Event Type
           IFM_Module_RobotArm:I1.Data[46].13   // Port 3 Event Type
           IFM_Module_RobotArm:I1.Data[46].14   // Port 3 Event Mode
           IFM_Module_RobotArm:I1.Data[46].15   // Port 3 Event Mode
           IFM_Module_RobotArm:I1.Data[46].2   // Port 3 Event Code 2
           IFM_Module_RobotArm:I1.Data[46].3   // Port 3 Event Code 2
           IFM_Module_RobotArm:I1.Data[46].4   // Port 3 Event Code 2
           IFM_Module_RobotArm:I1.Data[46].5   // Port 3 Event Code 2
           IFM_Module_RobotArm:I1.Data[46].6   // Port 3 Event Code 2
           IFM_Module_RobotArm:I1.Data[46].7   // Port 3 Event Code 2
           IFM_Module_RobotArm:I1.Data[46].11   // Port 3 Event Source
           IFM_Module_RobotArm:I1.Data[46].8   // Port 3 Event Instance
           IFM_Module_RobotArm:I1.Data[46].9   // Port 3 Event Instance
           IFM_Module_RobotArm:I1.Data[47].0   // Port 3 Event Code 1
           IFM_Module_RobotArm:I1.Data[47].1   // Port 3 Event Code 1
           IFM_Module_RobotArm:I1.Data[47]   // Port 3 IO-Link Event Data
           IFM_Module_RobotArm:I1.Data[47].10   // Port 3 Event Code 2
           IFM_Module_RobotArm:I1.Data[47].11   // Port 3 Event Code 2
           IFM_Module_RobotArm:I1.Data[47].12   // Port 3 Event Code 2
           IFM_Module_RobotArm:I1.Data[47].13   // Port 3 Event Code 2
           IFM_Module_RobotArm:I1.Data[47].14   // Port 3 Event Code 2
           IFM_Module_RobotArm:I1.Data[47].2   // Port 3 Event Code 1
           IFM_Module_RobotArm:I1.Data[47].3   // Port 3 Event Code 1
           IFM_Module_RobotArm:I1.Data[47].4   // Port 3 Event Code 1
           IFM_Module_RobotArm:I1.Data[47].5   // Port 3 Event Code 1
           IFM_Module_RobotArm:I1.Data[47].6   // Port 3 Event Code 1
           IFM_Module_RobotArm:I1.Data[47].7   // Port 3 Event Code 1
           IFM_Module_RobotArm:I1.Data[47].8   // Port 3 Event Code 2
           IFM_Module_RobotArm:I1.Data[47].9   // Port 3 Event Code 2
           IFM_Module_RobotArm:I1.Data[47].15   // Port 3 Event Code 2
           IFM_Module_RobotArm:I1.Data[48]   // Port 3 IO-Link Event Data
           IFM_Module_RobotArm:I1.Data[48].0   // Port 3 Event Instance
           IFM_Module_RobotArm:I1.Data[48].1   // Port 3 Event Instance
           IFM_Module_RobotArm:I1.Data[48].10   // Port 3 Event Code 1
           IFM_Module_RobotArm:I1.Data[48].11   // Port 3 Event Code 1
           IFM_Module_RobotArm:I1.Data[48].12   // Port 3 Event Code 1
           IFM_Module_RobotArm:I1.Data[48].13   // Port 3 Event Code 1
           IFM_Module_RobotArm:I1.Data[48].14   // Port 3 Event Code 1
           IFM_Module_RobotArm:I1.Data[48].15   // Port 3 Event Code 1
           IFM_Module_RobotArm:I1.Data[48].3   // Port 3 Event Source
           IFM_Module_RobotArm:I1.Data[41]   // Port 3 IO Link Status
           IFM_Module_RobotArm:I1.Data[45].4   // Port 3 Event Type
           IFM_Module_RobotArm:I1.Data[45].5   // Port 3 Event Type
           IFM_Module_RobotArm:I1.Data[45].6   // Port 3 Event Mode
           IFM_Module_RobotArm:I1.Data[48].8   // Port 3 Event Code 1
           IFM_Module_RobotArm:I1.Data[48].9   // Port 3 Event Code 1
           IFM_Module_RobotArm:I1.Data[48].2   // Port 3 Event Instance
           IFM_Module_RobotArm:I1.Data[49].0   // Port 3 Event Code 2
           IFM_Module_RobotArm:I1.Data[49].1   // Port 3 Event Code 2
           IFM_Module_RobotArm:I1.Data[49].10   // Reserved
           IFM_Module_RobotArm:I1.Data[49].11   // Reserved
           IFM_Module_RobotArm:I1.Data[49].12   // Reserved
           IFM_Module_RobotArm:I1.Data[49].13   // Reserved
           IFM_Module_RobotArm:I1.Data[49].14   // Reserved
           IFM_Module_RobotArm:I1.Data[49].15   // Reserved
           IFM_Module_RobotArm:I1.Data[49].2   // Port 3 Event Code 2
           IFM_Module_RobotArm:I1.Data[49].3   // Port 3 Event Code 2
           IFM_Module_RobotArm:I1.Data[49].4   // Port 3 Event Code 2
           IFM_Module_RobotArm:I1.Data[49].5   // Port 3 Event Code 2
           IFM_Module_RobotArm:I1.Data[49].6   // Port 3 Event Code 2
           IFM_Module_RobotArm:I1.Data[49].7   // Port 3 Event Code 2
           IFM_Module_RobotArm:I1.Data[49].8   // Reserved
           IFM_Module_RobotArm:I1.Data[49].9   // Reserved
           IFM_Module_RobotArm:I1.Data[4]   // SubIndex Number
           IFM_Module_RobotArm:I1.Data[45].7   // Port 3 Event Mode
           IFM_Module_RobotArm:I1.Data[50].0   // Port 4 IO-Link Mode
           IFM_Module_RobotArm:I1.Data[41].1   // Port 3 NO IO-Link Device Connected
           IFM_Module_RobotArm:I1.Data[50].10   // Reserved
           IFM_Module_RobotArm:I1.Data[50].11   // Reserved
           IFM_Module_RobotArm:I1.Data[50].12   // Reserved
           IFM_Module_RobotArm:I1.Data[50].13   // Reserved
           IFM_Module_RobotArm:I1.Data[50].14   // Reserved
           IFM_Module_RobotArm:I1.Data[50].15   // Reserved
           IFM_Module_RobotArm:I1.Data[50].2   // Port 4 IO-Link Data Invalid
           IFM_Module_RobotArm:I1.Data[50].3   // Port 4 Incorrect Vendor or Device ID
           IFM_Module_RobotArm:I1.Data[41].4   // Port 3 IO-Link Data String Error
           IFM_Module_RobotArm:I1.Data[50].5   // Reserved
           IFM_Module_RobotArm:I1.Data[50].6   // Reserved
           IFM_Module_RobotArm:I1.Data[50].7   // Reserved
           IFM_Module_RobotArm:I1.Data[50].8   // Reserved
           IFM_Module_RobotArm:I1.Data[50].9   // Reserved
           IFM_Module_RobotArm:I1.Data[51]   // Port 4 Vendor ID
           IFM_Module_RobotArm:I1.Data[52]   // Port 4 Device ID (Low Word)
           IFM_Module_RobotArm:I1.Data[53]   // Port 4 Device ID (High Word)
           IFM_Module_RobotArm:I1.Data[49]   // Port 3 IO-Link Event Data
           IFM_Module_RobotArm:I1.Data[54]   // Port 4 IO-Link Event Data
           IFM_Module_RobotArm:I1.Data[54].0   // Port 4 Event Instance
           IFM_Module_RobotArm:I1.Data[54].1   // Port 4 Event Instance
           IFM_Module_RobotArm:I1.Data[54].10   // Port 4 Event Code 1
           IFM_Module_RobotArm:I1.Data[54].11   // Port 4 Event Code 1
           IFM_Module_RobotArm:I1.Data[54].12   // Port 4 Event Code 1
           IFM_Module_RobotArm:I1.Data[54].13   // Port 4 Event Code 1
           IFM_Module_RobotArm:I1.Data[54].14   // Port 4 Event Code 1
           IFM_Module_RobotArm:I1.Data[54].15   // Port 4 Event Code 1
           IFM_Module_RobotArm:I1.Data[54].3   // Port 4 Event Source
           IFM_Module_RobotArm:I1.Data[48].4   // Port 3 Event Type
           IFM_Module_RobotArm:I1.Data[48].5   // Port 3 Event Type
           IFM_Module_RobotArm:I1.Data[48].6   // Port 3 Event Mode
           IFM_Module_RobotArm:I1.Data[48].7   // Port 3 Event Mode
           IFM_Module_RobotArm:I1.Data[54].8   // Port 4 Event Code 1
           IFM_Module_RobotArm:I1.Data[54].9   // Port 4 Event Code 1
           IFM_Module_RobotArm:I1.Data[46]   // Port 3 IO-Link Event Data
           IFM_Module_RobotArm:I1.Data[55].0   // Port 4 Event Code 2
           IFM_Module_RobotArm:I1.Data[55].1   // Port 4 Event Code 2
           IFM_Module_RobotArm:I1.Data[55]   // Port 4 IO-Link Event Data
           IFM_Module_RobotArm:I1.Data[54].2   // Port 4 Event Instance
           IFM_Module_RobotArm:I1.Data[55].12   // Port 4 Event Type
           IFM_Module_RobotArm:I1.Data[55].13   // Port 4 Event Type
           IFM_Module_RobotArm:I1.Data[55].14   // Port 4 Event Mode
           IFM_Module_RobotArm:I1.Data[55].15   // Port 4 Event Mode
           IFM_Module_RobotArm:I1.Data[55].2   // Port 4 Event Code 2
           IFM_Module_RobotArm:I1.Data[55].3   // Port 4 Event Code 2
           IFM_Module_RobotArm:I1.Data[55].4   // Port 4 Event Code 2
           IFM_Module_RobotArm:I1.Data[55].5   // Port 4 Event Code 2
           IFM_Module_RobotArm:I1.Data[55].6   // Port 4 Event Code 2
           IFM_Module_RobotArm:I1.Data[55].7   // Port 4 Event Code 2
           IFM_Module_RobotArm:I1.Data[55].11   // Port 4 Event Source
           IFM_Module_RobotArm:I1.Data[55].8   // Port 4 Event Instance
           IFM_Module_RobotArm:I1.Data[55].9   // Port 4 Event Instance
           IFM_Module_RobotArm:I1.Data[56].0   // Port 4 Event Code 1
           IFM_Module_RobotArm:I1.Data[56].1   // Port 4 Event Code 1
           IFM_Module_RobotArm:I1.Data[56]   // Port 4 IO-Link Event Data
           IFM_Module_RobotArm:I1.Data[56].10   // Port 4 Event Code 2
           IFM_Module_RobotArm:I1.Data[56].11   // Port 4 Event Code 2
           IFM_Module_RobotArm:I1.Data[56].12   // Port 4 Event Code 2
           IFM_Module_RobotArm:I1.Data[56].13   // Port 4 Event Code 2
           IFM_Module_RobotArm:I1.Data[56].14   // Port 4 Event Code 2
           IFM_Module_RobotArm:I1.Data[56].2   // Port 4 Event Code 1
           IFM_Module_RobotArm:I1.Data[56].3   // Port 4 Event Code 1
           IFM_Module_RobotArm:I1.Data[56].4   // Port 4 Event Code 1
           IFM_Module_RobotArm:I1.Data[56].5   // Port 4 Event Code 1
           IFM_Module_RobotArm:I1.Data[56].6   // Port 4 Event Code 1
           IFM_Module_RobotArm:I1.Data[56].7   // Port 4 Event Code 1
           IFM_Module_RobotArm:I1.Data[56].8   // Port 4 Event Code 2
           IFM_Module_RobotArm:I1.Data[56].9   // Port 4 Event Code 2
           IFM_Module_RobotArm:I1.Data[56].15   // Port 4 Event Code 2
           IFM_Module_RobotArm:I1.Data[57]   // Port 4 IO-Link Event Data
           IFM_Module_RobotArm:I1.Data[57].0   // Port 4 Event Instance
           IFM_Module_RobotArm:I1.Data[57].1   // Port 4 Event Instance
           IFM_Module_RobotArm:I1.Data[57].10   // Port 4 Event Code 1
           IFM_Module_RobotArm:I1.Data[57].11   // Port 4 Event Code 1
           IFM_Module_RobotArm:I1.Data[57].12   // Port 4 Event Code 1
           IFM_Module_RobotArm:I1.Data[57].13   // Port 4 Event Code 1
           IFM_Module_RobotArm:I1.Data[57].14   // Port 4 Event Code 1
           IFM_Module_RobotArm:I1.Data[57].15   // Port 4 Event Code 1
           IFM_Module_RobotArm:I1.Data[57].3   // Port 4 Event Source
           IFM_Module_RobotArm:I1.Data[50]   // Port 4 IO Link Status
           IFM_Module_RobotArm:I1.Data[54].4   // Port 4 Event Type
           IFM_Module_RobotArm:I1.Data[54].5   // Port 4 Event Type
           IFM_Module_RobotArm:I1.Data[54].6   // Port 4 Event Mode
           IFM_Module_RobotArm:I1.Data[57].8   // Port 4 Event Code 1
           IFM_Module_RobotArm:I1.Data[57].9   // Port 4 Event Code 1
           IFM_Module_RobotArm:I1.Data[57].2   // Port 4 Event Instance
           IFM_Module_RobotArm:I1.Data[58].0   // Port 4 Event Code 2
           IFM_Module_RobotArm:I1.Data[58].1   // Port 4 Event Code 2
           IFM_Module_RobotArm:I1.Data[58].10   // Reserved
           IFM_Module_RobotArm:I1.Data[58].11   // Reserved
           IFM_Module_RobotArm:I1.Data[58].12   // Reserved
           IFM_Module_RobotArm:I1.Data[58].13   // Reserved
           IFM_Module_RobotArm:I1.Data[58].14   // Reserved
           IFM_Module_RobotArm:I1.Data[58].15   // Reserved
           IFM_Module_RobotArm:I1.Data[58].2   // Port 4 Event Code 2
           IFM_Module_RobotArm:I1.Data[58].3   // Port 4 Event Code 2
           IFM_Module_RobotArm:I1.Data[58].4   // Port 4 Event Code 2
           IFM_Module_RobotArm:I1.Data[58].5   // Port 4 Event Code 2
           IFM_Module_RobotArm:I1.Data[58].6   // Port 4 Event Code 2
           IFM_Module_RobotArm:I1.Data[58].7   // Port 4 Event Code 2
           IFM_Module_RobotArm:I1.Data[58].8   // Reserved
           IFM_Module_RobotArm:I1.Data[58].9   // Reserved
           IFM_Module_RobotArm:I1.Data[58]   // Port 4 IO-Link Event Data
           IFM_Module_RobotArm:I1.Data[6].10   // Command Response or Diagnostic Data 0
           IFM_Module_RobotArm:I1.Data[50].1   // Port 4 NO IO-Link Device Connected
           IFM_Module_RobotArm:I1.Data[5].1   // TRUE if Write Acyclic Command Response
           IFM_Module_RobotArm:I1.Data[5].10   // Target Mode
           IFM_Module_RobotArm:I1.Data[5].11   // Target Mode
           IFM_Module_RobotArm:I1.Data[5].12   // Target Mode
           IFM_Module_RobotArm:I1.Data[5].13   // Target Mode
           IFM_Module_RobotArm:I1.Data[5].14   // Target Mode
           IFM_Module_RobotArm:I1.Data[5].15   // Target Mode
           IFM_Module_RobotArm:I1.Data[5].2   // Reserved
           IFM_Module_RobotArm:I1.Data[5].3   // Reserved
           IFM_Module_RobotArm:I1.Data[5].4   // Reserved
           IFM_Module_RobotArm:I1.Data[5].5   // Reserved
           IFM_Module_RobotArm:I1.Data[5].6   // Reserved
           IFM_Module_RobotArm:I1.Data[5].7   // TRUE if HandShake Response To Acyclic Command
           IFM_Module_RobotArm:I1.Data[5].8   // Target Mode
           IFM_Module_RobotArm:I1.Data[5].9   // Target Mode
           IFM_Module_RobotArm:I1.Data[59]   // Port 1 Input Process Data
           IFM_Module_RobotArm:I1.Data[60]   // Port 1 Input Process Data
           IFM_Module_RobotArm:I1.Data[61]   // Port 1 Input Process Data
           IFM_Module_RobotArm:I1.Data[62]   // Port 1 Input Process Data
           IFM_Module_RobotArm:I1.Data[63]   // Port 1 Input Process Data
           IFM_Module_RobotArm:I1.Data[64]   // Port 1 Input Process Data
           IFM_Module_RobotArm:I1.Data[65]   // Port 1 Input Process Data
           IFM_Module_RobotArm:I1.Data[66]   // Port 1 Input Process Data
           IFM_Module_RobotArm:I1.Data[67]   // Port 1 Input Process Data
           IFM_Module_RobotArm:I1.Data[68]   // Port 1 Input Process Data
           IFM_Module_RobotArm:I1.Data[6]   // Command Response Byte Length & Command Response or Diagnostic Data 0
           IFM_Module_RobotArm:I1.Data[55].10   // Port 4 Event Instance
           IFM_Module_RobotArm:I1.Data[6].0   // Command Byte Length Bit 0
           IFM_Module_RobotArm:I1.Data[6].11   // Command Response or Diagnostic Data 0
           IFM_Module_RobotArm:I1.Data[6].12   // Command Response or Diagnostic Data 0
           IFM_Module_RobotArm:I1.Data[6].13   // Command Response or Diagnostic Data 0
           IFM_Module_RobotArm:I1.Data[6].14   // Command Response or Diagnostic Data 0
           IFM_Module_RobotArm:I1.Data[6].15   // Command Response or Diagnostic Data 0
           IFM_Module_RobotArm:I1.Data[6].9   // Command Response or Diagnostic Data 0
           IFM_Module_RobotArm:I1.Data[6].1   // Command Byte Length Bit 1
           IFM_Module_RobotArm:I1.Data[6].2   // Command Byte Length Bit 2
           IFM_Module_RobotArm:I1.Data[6].3   // Command Byte Length Bit 3
           IFM_Module_RobotArm:I1.Data[6].4   // Command Byte Length Bit 4
           IFM_Module_RobotArm:I1.Data[6].5   // Command Byte Length Bit 5
           IFM_Module_RobotArm:I1.Data[6].6   // Command Byte Length Bit 6
           IFM_Module_RobotArm:I1.Data[50].4   // Port 4 IO-Link Data String Error
           IFM_Module_RobotArm:I1.Data[5].0   // TRUE if Read Acyclic Command Response
           IFM_Module_RobotArm:I1.Data[69]   // Port 1 Input Process Data
           IFM_Module_RobotArm:I1.Data[70]   // Port 1 Input Process Data
           IFM_Module_RobotArm:I1.Data[71]   // Port 1 Input Process Data
           IFM_Module_RobotArm:I1.Data[72]   // Port 1 Input Process Data
           IFM_Module_RobotArm:I1.Data[73]   // Port 1 Input Process Data
           IFM_Module_RobotArm:I1.Data[74]   // Port 1 Input Process Data
           IFM_Module_RobotArm:I1.Data[75]   // Port 2 Input Process Data
           IFM_Module_RobotArm:I1.Data[76]   // Port 2 Input Process Data
           IFM_Module_RobotArm:I1.Data[77]   // Port 2 Input Process Data
           IFM_Module_RobotArm:I1.Data[78]   // Port 2 Input Process Data
           IFM_Module_RobotArm:I1.Data[8]   // Command Response Or Diagnostic Data 3
           IFM_Module_RobotArm:I1.Data[79]   // Port 2 Input Process Data
           IFM_Module_RobotArm:I1.Data[80]   // Port 2 Input Process Data
           IFM_Module_RobotArm:I1.Data[81]   // Port 2 Input Process Data
           IFM_Module_RobotArm:I1.Data[82]   // Port 2 Input Process Data
           IFM_Module_RobotArm:I1.Data[83]   // Port 2 Input Process Data
           IFM_Module_RobotArm:I1.Data[84]   // Port 2 Input Process Data
           IFM_Module_RobotArm:I1.Data[85]   // Port 2 Input Process Data
           IFM_Module_RobotArm:I1.Data[86]   // Port 2 Input Process Data
           IFM_Module_RobotArm:I1.Data[87]   // Port 2 Input Process Data
           IFM_Module_RobotArm:I1.Data[88]   // Port 2 Input Process Data
           IFM_Module_RobotArm:I1.Data[9]   // Command Response Or Diagnostic Data 5
           IFM_Module_RobotArm:I1.Data[89]   // Port 2 Input Process Data
           IFM_Module_RobotArm:I1.Data[90]   // Port 2 Input Process Data
           IFM_Module_RobotArm:I1.Data[91]   // Port 3 Input Process Data
           IFM_Module_RobotArm:I1.Data[92]   // Port 3 Input Process Data
           IFM_Module_RobotArm:I1.Data[93]   // Port 3 Input Process Data
           IFM_Module_RobotArm:I1.Data[94]   // Port 3 Input Process Data
           IFM_Module_RobotArm:I1.Data[95]   // Port 3 Input Process Data
           IFM_Module_RobotArm:I1.Data[96]   // Port 3 Input Process Data
           IFM_Module_RobotArm:I1.Data[97]   // Port 3 Input Process Data
           IFM_Module_RobotArm:I1.Data[98]   // Port 3 Input Process Data
           IFM_Module_RobotArm:I1.Data[99]   // Port 3 Input Process Data
           IFM_Module_RobotArm:I1.Data[6].8   // Command Response or Diagnostic Data 0
           IFM_Module_RobotArm:I1.Data[54].7   // Port 4 Event Mode
           IFM_Module_RobotArm:I1.Data[57].4   // Port 4 Event Type
           IFM_Module_RobotArm:I1.Data[6].7   // Command Byte Length Bit 7
           IFM_Module_RobotArm:I1.Data[57].5   // Port 4 Event Type
           IFM_Module_RobotArm:I1.Data[57].6   // Port 4 Event Mode
           IFM_Module_RobotArm:I1.Data[57].7   // Port 4 Event Mode
           IFM_Module_RobotArm:I1.Data[5]   // Read/Write Command Code; HandShake; Command Result
           IFM_Module_RobotArm:O1.Data[0].0   // Port 1 Pin 4 Digital Output
           IFM_Module_RobotArm:O1.Data[0].1   // Port 2 Pin 4 Digital Output
           IFM_Module_RobotArm:O1.Data[0].10   // Reserved
           IFM_Module_RobotArm:O1.Data[0].11   // Reserved
           IFM_Module_RobotArm:O1.Data[0].12   // Reserved
           IFM_Module_RobotArm:O1.Data[0].13   // Reserved
           IFM_Module_RobotArm:O1.Data[0].14   // Reserved
           IFM_Module_RobotArm:O1.Data[0].15   // Reserved
           IFM_Module_RobotArm:O1.Data[0].2   // Port 3 Pin 4 Digital Output
           IFM_Module_RobotArm:O1.Data[0].3   // Port 4 Pin 4 Digital Output
           IFM_Module_RobotArm:O1.Data[0].4   // Reserved
           IFM_Module_RobotArm:O1.Data[0].5   // Reserved
           IFM_Module_RobotArm:O1.Data[0].6   // Reserved
           IFM_Module_RobotArm:O1.Data[0].7   // Reserved
           IFM_Module_RobotArm:O1.Data[0].8   // Reserved
           IFM_Module_RobotArm:O1.Data[0].9   // Reserved
           IFM_Module_RobotArm:O1.Data[10]   // Command Data Array 8
           IFM_Module_RobotArm:O1.Data[11]   // Command Data Array 10
           IFM_Module_RobotArm:O1.Data[12]   // Command Data Array 12
           IFM_Module_RobotArm:O1.Data[13]   // Command Data Array 14
           IFM_Module_RobotArm:O1.Data[14]   // Command Data Array 16
           IFM_Module_RobotArm:O1.Data[1]   // Reserved
           IFM_Module_RobotArm:O1.Data[15]   // Command Data Array 18
           IFM_Module_RobotArm:O1.Data[16]   // Command Data Array 20
           IFM_Module_RobotArm:O1.Data[22]   // Reserved
           IFM_Module_RobotArm:O1.Data[23]   // Port 1 Digital Output Process Data
           IFM_Module_RobotArm:O1.Data[24]   // Port 1 Digital Output Process Data
           IFM_Module_RobotArm:O1.Data[25]   // Port 1 Digital Output Process Data
           IFM_Module_RobotArm:O1.Data[26]   // Port 1 Digital Output Process Data
           IFM_Module_RobotArm:O1.Data[27]   // Port 1 Digital Output Process Data
           IFM_Module_RobotArm:O1.Data[28]   // Port 1 Digital Output Process Data
           IFM_Module_RobotArm:O1.Data[29]   // Port 1 Digital Output Process Data
           IFM_Module_RobotArm:O1.Data[2]   // AL1x2x Port Number
           IFM_Module_RobotArm:O1.Data[30]   // Port 1 Digital Output Process Data
           IFM_Module_RobotArm:O1.Data[31]   // Port 1 Digital Output Process Data
           IFM_Module_RobotArm:O1.Data[32]   // Port 1 Digital Output Process Data
           IFM_Module_RobotArm:O1.Data[33]   // Port 1 Digital Output Process Data
           IFM_Module_RobotArm:O1.Data[34]   // Port 1 Digital Output Process Data
           IFM_Module_RobotArm:O1.Data[35]   // Port 1 Digital Output Process Data
           IFM_Module_RobotArm:O1.Data[36]   // Port 1 Digital Output Process Data
           IFM_Module_RobotArm:O1.Data[37]   // Port 1 Digital Output Process Data
           IFM_Module_RobotArm:O1.Data[38]   // Port 1 Digital Output Process Data
           IFM_Module_RobotArm:O1.Data[39]   // Port 2 Digital Output Process Data
           IFM_Module_RobotArm:O1.Data[3]   // Index Number
           IFM_Module_RobotArm:O1.Data[40]   // Port 2 Digital Output Process Data
           IFM_Module_RobotArm:O1.Data[41]   // Port 2 Digital Output Process Data
           IFM_Module_RobotArm:O1.Data[42]   // Port 2 Digital Output Process Data
           IFM_Module_RobotArm:O1.Data[43]   // Port 2 Digital Output Process Data
           IFM_Module_RobotArm:O1.Data[44]   // Port 2 Digital Output Process Data
           IFM_Module_RobotArm:O1.Data[45]   // Port 2 Digital Output Process Data
           IFM_Module_RobotArm:O1.Data[46]   // Port 2 Digital Output Process Data
           IFM_Module_RobotArm:O1.Data[47]   // Port 2 Digital Output Process Data
           IFM_Module_RobotArm:O1.Data[48]   // Port 2 Digital Output Process Data
           IFM_Module_RobotArm:O1.Data[49]   // Port 2 Digital Output Process Data
           IFM_Module_RobotArm:O1.Data[4]   // SubIndex Number
           IFM_Module_RobotArm:O1.Data[50]   // Port 2 Digital Output Process Data
           IFM_Module_RobotArm:O1.Data[51]   // Port 2 Digital Output Process Data
           IFM_Module_RobotArm:O1.Data[52]   // Port 2 Digital Output Process Data
           IFM_Module_RobotArm:O1.Data[53]   // Port 2 Digital Output Process Data
           IFM_Module_RobotArm:O1.Data[54]   // Port 2 Digital Output Process Data
           IFM_Module_RobotArm:O1.Data[55]   // Port 3 Digital Output Process Data
           IFM_Module_RobotArm:O1.Data[56]   // Port 3 Digital Output Process Data
           IFM_Module_RobotArm:O1.Data[57]   // Port 3 Digital Output Process Data
           IFM_Module_RobotArm:O1.Data[58]   // Port 3 Digital Output Process Data
           IFM_Module_RobotArm:O1.Data[59]   // Port 3 Digital Output Process Data
           IFM_Module_RobotArm:O1.Data[5]   // Read/Write Command Code; Trigger Bit; Command Byte Length
           IFM_Module_RobotArm:O1.Data[5].0   // Set TRUE to Read
           IFM_Module_RobotArm:O1.Data[5].10   // Command Byte Length Bit 2
           IFM_Module_RobotArm:O1.Data[5].11   // Command Byte Length Bit 3
           IFM_Module_RobotArm:O1.Data[5].12   // Command Byte Length Bit 4
           IFM_Module_RobotArm:O1.Data[5].13   // Command Byte Length Bit 5
           IFM_Module_RobotArm:O1.Data[5].14   // Command Byte Length Bit 6
           IFM_Module_RobotArm:O1.Data[5].15   // Command Byte Length Bit 7
           IFM_Module_RobotArm:O1.Data[5].2   // Reserved
           IFM_Module_RobotArm:O1.Data[5].3   // Reserved
           IFM_Module_RobotArm:O1.Data[5].4   // Reserved
           IFM_Module_RobotArm:O1.Data[5].5   // Reserved
           IFM_Module_RobotArm:O1.Data[5].6   // Reserved
           IFM_Module_RobotArm:O1.Data[5].8   // Command Byte Length Bit 0
           IFM_Module_RobotArm:O1.Data[5].9   // Command Byte Length Bit 1
           IFM_Module_RobotArm:O1.Data[60]   // Port 3 Digital Output Process Data
           IFM_Module_RobotArm:O1.Data[61]   // Port 3 Digital Output Process Data
           IFM_Module_RobotArm:O1.Data[62]   // Port 3 Digital Output Process Data
           IFM_Module_RobotArm:O1.Data[63]   // Port 3 Digital Output Process Data
           IFM_Module_RobotArm:O1.Data[64]   // Port 3 Digital Output Process Data
           IFM_Module_RobotArm:O1.Data[65]   // Port 3 Digital Output Process Data
           IFM_Module_RobotArm:O1.Data[66]   // Port 3 Digital Output Process Data
           IFM_Module_RobotArm:O1.Data[67]   // Port 3 Digital Output Process Data
           IFM_Module_RobotArm:O1.Data[68]   // Port 3 Digital Output Process Data
           IFM_Module_RobotArm:O1.Data[69]   // Port 3 Digital Output Process Data
           IFM_Module_RobotArm:O1.Data[6]   // Command Data Array 0
           IFM_Module_RobotArm:O1.Data[70]   // Port 3 Digital Output Process Data
           IFM_Module_RobotArm:O1.Data[71]   // Port 4 Digital Output Process Data
           IFM_Module_RobotArm:O1.Data[72]   // Port 4 Digital Output Process Data
           IFM_Module_RobotArm:O1.Data[73]   // Port 4 Digital Output Process Data
           IFM_Module_RobotArm:O1.Data[74]   // Port 4 Digital Output Process Data
           IFM_Module_RobotArm:O1.Data[75]   // Port 4 Digital Output Process Data
           IFM_Module_RobotArm:O1.Data[76]   // Port 4 Digital Output Process Data
           IFM_Module_RobotArm:O1.Data[77]   // Port 4 Digital Output Process Data
           IFM_Module_RobotArm:O1.Data[78]   // Port 4 Digital Output Process Data
           IFM_Module_RobotArm:O1.Data[79]   // Port 4 Digital Output Process Data
           IFM_Module_RobotArm:O1.Data[7]   // Command Data Array 2
           IFM_Module_RobotArm:O1.Data[80]   // Port 4 Digital Output Process Data
           IFM_Module_RobotArm:O1.Data[81]   // Port 4 Digital Output Process Data
           IFM_Module_RobotArm:O1.Data[82]   // Port 4 Digital Output Process Data
           IFM_Module_RobotArm:O1.Data[83]   // Port 4 Digital Output Process Data
           IFM_Module_RobotArm:O1.Data[84]   // Port 4 Digital Output Process Data
           IFM_Module_RobotArm:O1.Data[85]   // Port 4 Digital Output Process Data
           IFM_Module_RobotArm:O1.Data[86]   // Port 4 Digital Output Process Data
           IFM_Module_RobotArm:O1.Data[8]   // Command Data Array 4
           IFM_Module_RobotArm:O1.Data[9]   // Command Data Array 6
           IFM_Module_RobotArm:O1.Data[5].7   // Trigger Acyclic Command
           IFM_Module_RobotArm:O1.Data[17]   // Command Data Array 22
           IFM_Module_RobotArm:O1.Data[18]   // Command Data Array 24
           IFM_Module_RobotArm:O1.Data[19]   // Command Data Array 26
           IFM_Module_RobotArm:O1.Data[20]   // Command Data Array 28
           IFM_Module_RobotArm:O1.Data[21]   // Command Data Array 30
           IFM_Module_RobotArm:O1.Data[0]   // AL1x2x Digital Output Status
           IFM_Module_RobotArm:O1.Data[5].1   // Set TRUE to Write
END_MODULES
